(* IEC 61131-3 sources: ElnaAutomator/ExampleProject/build_USO_ecl, 1 file *)

(* ---- plc.st ---- *)
TYPE
  struct_singleOutput : STRUCT
    wait_time : TIME;
    inCommand : WORD;
    inOpcCommandsDisabled : BOOL;
    Q : BOOL;
    status : DWORD;
    OpcCommandsDisabled : BOOL;
    inCommand_Alg : WORD;
    inCommand_ARM : WORD;
  END_STRUCT;
  Im_singleOutputs : STRUCT
    So0 : struct_singleOutput;
    So1 : struct_singleOutput;
    So2 : struct_singleOutput;
    So3 : struct_singleOutput;
    So4 : struct_singleOutput;
    So5 : struct_singleOutput;
    So6 : struct_singleOutput;
    So7 : struct_singleOutput;
  END_STRUCT;
  struct_SectionSwitch : STRUCT
    inCommand : WORD;
    status : DWORD;
    onStatus : BYTE;
    inOpcCommandsDisabled : BOOL;
    sdvig : BOOL;
    Ns : BOOL;
    CommandFault : BOOL;
    Accident : BOOL;
    Local : BOOL;
    Distance : BOOL;
    OpcCommandsDisabled : BOOL;
    lastCmdIsOn : BOOL;
    offKNA : BOOL;
    basketStatus : BYTE;
    ISVALIDREF_statOn : BOOL;
    ISVALIDREF_statOff : BOOL;
    ISVALIDREF_cmdOn : BOOL;
    ISVALIDREF_cmdOff : BOOL;
    ISVALIDREF_inBreakCmdOn : BOOL;
    ISVALIDREF_inBreakCmdOff : BOOL;
    BreakCmdOn : BOOL;
    BreakCmdOff : BOOL;
    ISVALIDREF_basketRolledIn : BOOL;
    ISVALIDREF_basketRolledOut : BOOL;
    ISVALIDREF_basketTest : BOOL;
    inCommand_Alg : WORD;
    inCommand_ARM : WORD;
    cmdOn : BOOL;
    cmdOff : BOOL;
    reliability : BOOL;
  END_STRUCT;
  TYPE_ReliableBit : STRUCT
    value : BOOL;
    reliability : BOOL;
    _inversed : BOOL;
  END_STRUCT;
  struct_DI : STRUCT
    imit : BOOL;
    value : WORD;
    reliability : WORD;
    bits : ARRAY [0..15] OF TYPE_ReliableBit;
    blConnect : BOOL;
  END_STRUCT;
  DiConfig : STRUCT
    Di : struct_DI;
    Di1 : struct_DI;
    Di2 : struct_DI;
    Di3 : struct_DI;
    Di4 : struct_DI;
  END_STRUCT;
  TYPE_ProtectionTags : STRUCT
    NOTHING : BYTE := 0;
    AOB : BYTE := 1;
    AOS : BYTE := 2;
    AOPOJ : BYTE := 3;
  END_STRUCT;
  struct_singleSignal : STRUCT
    reliability : BOOL;
    inverse : BOOL;
    DelayOn : TIME;
    DelayOff : TIME;
    Q : BOOL;
    status : DWORD;
    Disabled_Sig : BOOL;
  END_STRUCT;
  struct_AiProtection : STRUCT
    controlLimit : BYTE;
    delay : TIME;
    inTag : BYTE;
    inRunOnStart : BOOL;
    inCanRun : BOOL;
    inOpcCommandsDisabled : BOOL;
    inCommand : WORD;
    inCommand_Alg : WORD;
    inCommand_ARM : WORD;
    Tag : BYTE;
    status : DWORD;
    CanRun : BOOL;
    OpcCommandsDisabled : BOOL;
    isRunning : BOOL;
    HasError : BOOL;
    isEnded : BOOL;
    Remont : BOOL;
    Check : BOOL;
    Signaling : BOOL;
    SignalingTP : BOOL;
    RunOnStart : BOOL;
  END_STRUCT;
  TDoubleData : STRUCT
    wFlags : UINT := 0;
    dblValue : LREAL := 0.0;
  END_STRUCT;
  struct_DO : STRUCT
    imit : BOOL;
    blConnect : BOOL;
    value : WORD;
    bits : ARRAY [0..15] OF BOOL;
  END_STRUCT;
  DoConfig : STRUCT
    Do1 : struct_DO;
    Do2 : struct_DO;
    Do3 : struct_DO;
    Do4 : struct_DO;
    Do5 : struct_DO;
  END_STRUCT;
  struct_ReserveIM2 : STRUCT
    var1 : BOOL;
    var2 : BOOL;
  END_STRUCT;
  struct_Kran : STRUCT
    inCommand : WORD;
    status : DWORD;
    onStatus : BYTE;
    inOpcCommandsDisabled : BOOL;
    sdvig : BOOL;
    Ns : BOOL;
    Dp : BOOL;
    CommandFault : BOOL;
    Accident : BOOL;
    Auto : BOOL;
    Manual : BOOL;
    Local : BOOL;
    Distance : BOOL;
    ErrorPowerOff : BOOL;
    ErrorBlock : BOOL;
    So : BOOL;
    Sz : BOOL;
    OpcCommandsDisabled : BOOL;
    lastCmdIsOn : BOOL;
    ISVALIDREF_statOn : BOOL;
    ISVALIDREF_statOff : BOOL;
    ISVALIDREF_cmdOn : BOOL;
    ISVALIDREF_cmdOff : BOOL;
    ISVALIDREF_inSo : BOOL;
    ISVALIDREF_inSz : BOOL;
    ISVALIDREF_inDp : BOOL;
    continueHoldCommand : TIME;
    inCommand_Alg : WORD;
    inCommand_ARM : WORD;
    cmdOn : BOOL;
    cmdOff : BOOL;
    reliability : BOOL;
  END_STRUCT;
  struct_OilPump : STRUCT
    inCommand : WORD;
    inCommand_Alg : WORD;
    inCommand_ARM : WORD;
    status : DWORD;
    onStatus : BYTE;
    inOpcCommandsDisabled : BOOL;
    sdvig : BOOL;
    Ns : BOOL;
    CommandFault : BOOL;
    Accident : BOOL;
    Local : BOOL;
    Distance : BOOL;
    BreakCmdOn : BOOL;
    BreakCmdOff : BOOL;
    OpcCommandsDisabled : BOOL;
    lastCmdIsOn : BOOL;
    ISVALIDREF_statOn : BOOL;
    ISVALIDREF_statOff : BOOL;
    ISVALIDREF_cmdOn : BOOL;
    ISVALIDREF_cmdOff : BOOL;
    ISVALIDREF_inBreakCmdOn : BOOL;
    ISVALIDREF_inBreakCmdOff : BOOL;
    inBlocked : BOOL;
    Blocked : BOOL;
    Osnovnoy : BOOL;
    Rezervny : BOOL;
    cmdOn : BOOL;
    cmdOff : BOOL;
    reliability : BOOL;
  END_STRUCT;
  struct_Switch : STRUCT
    inCommand : WORD;
    status : DWORD;
    onStatus : BYTE;
    inOpcCommandsDisabled : BOOL;
    sdvig : BOOL;
    Ns : BOOL;
    CommandFault : BOOL;
    Accident : BOOL;
    Auto : BOOL;
    Manual : BOOL;
    Local : BOOL;
    Distance : BOOL;
    ErrorPowerOff : BOOL;
    ErrorBlock : BOOL;
    BreakCmdOn : BOOL;
    BreakCmdOff : BOOL;
    OpcCommandsDisabled : BOOL;
    lastCmdIsOn : BOOL;
    ISVALIDREF_statOn : BOOL;
    ISVALIDREF_statOff : BOOL;
    ISVALIDREF_cmdOn : BOOL;
    ISVALIDREF_cmdOff : BOOL;
    ISVALIDREF_inBreakCmdOn : BOOL;
    ISVALIDREF_inBreakCmdOff : BOOL;
    inCommand_Alg : WORD;
    inCommand_ARM : WORD;
    cmdOn : BOOL;
    cmdOff : BOOL;
    reliability : BOOL;
  END_STRUCT;
  Im_singleSignals : STRUCT
    SI0 : struct_singleSignal;
    SI1 : struct_singleSignal;
    SI2 : struct_singleSignal;
    SI3 : struct_singleSignal;
    SI4 : struct_singleSignal;
    SI5 : struct_singleSignal;
    SI6 : struct_singleSignal;
  END_STRUCT;
  ImConfig : STRUCT
    Kran1 : struct_Kran;
    Kran4 : struct_Kran;
    Kran2 : struct_Kran;
    Kran3 : struct_Kran;
    Nu : struct_OilPump;
    Nu2 : struct_OilPump;
    Avom1 : struct_Switch;
    Avom2 : struct_Switch;
    Avom3 : struct_Switch;
    Avom4 : struct_Switch;
    Mv : struct_SectionSwitch;
    SectionSwitch1 : struct_SectionSwitch;
    SingleSignals : Im_singleSignals;
    SingleOutputs : Im_singleOutputs;
  END_STRUCT;
  struct_DiProtection : STRUCT
    delay : TIME;
    inTag : BYTE;
    inRunOnStart : BOOL;
    inCanRun : BOOL;
    inOpcCommandsDisabled : BOOL;
    inCommand : WORD;
    inCommand_Alg : WORD;
    inCommand_ARM : WORD;
    Tag : BYTE;
    status : DWORD;
    CanRun : BOOL;
    OpcCommandsDisabled : BOOL;
    isRunning : BOOL;
    HasError : BOOL;
    isEnded : BOOL;
    Remont : BOOL;
    Check : BOOL;
    Signaling : BOOL;
    SignalingTP : BOOL;
    RunOnStart : BOOL;
  END_STRUCT;
  ProtectionsConfig : STRUCT
    Ap1 : struct_AiProtection;
    AiP1 : struct_AiProtection;
    AiP2 : struct_AiProtection;
    AiP3 : struct_AiProtection;
    DiP1 : struct_DiProtection;
    DiP2 : struct_DiProtection;
    DiP3 : struct_DiProtection;
    DiP4 : struct_DiProtection;
    DiP5 : struct_DiProtection;
  END_STRUCT;
  TYPE_StatusAi : STRUCT
    NOTDEFINED : BYTE := 0;
    LL : BYTE := 1;
    HL : BYTE := 2;
    NOTRELIABLE : BYTE := 3;
    normal : BYTE := 4;
    LW : BYTE := 5;
    HW : BYTE := 6;
    LA : BYTE := 7;
    HA : BYTE := 8;
  END_STRUCT;
  TItemAIN : STRUCT
    wFlags : UINT := 0;
    wReserved : UINT := 0;
    dblValue : LREAL := 0.0;
    nanosec : ULINT := 0;
    reserve : ULINT := 0;
  END_STRUCT;
  TItemDIN : STRUCT
    wFlags : UINT := 0;
    wValue : UINT := 0;
    nanosec : ULINT := 0;
    reserve : ULINT := 0;
  END_STRUCT;
  struct_AI : STRUCT
    value : LREAL;
    status : DWORD;
    interval : BYTE;
    inCommand : WORD;
    blConnect : BOOL;
    dLL : LREAL;
    dHL : LREAL;
    dLA : LREAL;
    dHA : LREAL;
    dLW : LREAL;
    dHW : LREAL;
    LL : LREAL;
    HL : LREAL;
    LA : LREAL;
    HA : LREAL;
    LW : LREAL;
    HW : LREAL;
    ISVALIDREF_LA : BOOL;
    ISVALIDREF_HA : BOOL;
    ISVALIDREF_LW : BOOL;
    ISVALIDREF_HW : BOOL;
    inpLL : LREAL;
    inpHL : LREAL;
    CurrentShotCircuit : LREAL;
    CurrentBreakCircuit : LREAL;
    maxChangeSpeed : LREAL;
    maxChangeSpeedDown : LREAL;
    ChangeSpeed : LREAL;
    histeresis : LREAL;
    aperturFilter : LREAL;
    exponentialFilter : LREAL;
    rassoglasovanie : LREAL;
    OpcCommandsDisabled : BOOL;
    Disabled_LA : BOOL;
    Disabled_HA : BOOL;
    Disabled_LW : BOOL;
    Disabled_HW : BOOL;
    delayLA : TIME;
    delayLW : TIME;
    delayHW : TIME;
    delayHA : TIME;
    minValue_ISVALIDREF : BOOL;
    maxValue_ISVALIDREF : BOOL;
    minValue : LREAL;
    maxValue : LREAL;
    inOpcCommandsDisabled : BOOL;
    imit : BOOL;
    remont : BOOL;
    NS : BOOL;
    NS_Min : BOOL;
    NS_Max : BOOL;
    inCommand_Alg : WORD;
    inCommand_ARM : WORD;
  END_STRUCT;
  AiConfig : STRUCT
    A1 : struct_AI;
    A2 : struct_AI;
  END_STRUCT;
  TWordData : STRUCT
    wFlags : UINT := 0;
    wValue : UINT := 0;
  END_STRUCT;
  TYPE_statusDualInput : STRUCT
    STATUS_NOTDEFINED : BYTE := 0;
    STATUS_ON : BYTE := 1;
    STATUS_OFF : BYTE := 2;
    STATUS_TRANSITIONAL : BYTE := 3;
    STATUS_ERROR : BYTE := 4;
  END_STRUCT;
  TYPE_AnalogLimitFlags : STRUCT
    NONE : BYTE := 0;
    LL : BYTE := 16#1;
    LW : BYTE := 16#2;
    HW : BYTE := 16#4;
    LA : BYTE := 16#8;
    HA : BYTE := 16#10;
    HL : BYTE := 16#20;
  END_STRUCT;
  TYPE_basketStats : STRUCT
    BASKET_NOTDEFINED : BYTE := 0;
    BASKET_ROLLEDIN : BYTE := 1;
    BASKET_ROLLEDOUT : BYTE := 2;
    BASKET_TRANSITIONAL : BYTE := 3;
    BASKET_ERROR : BYTE := 4;
    BASKET_TEST : BYTE := 5;
  END_STRUCT;
  TYPE_CommandAnalog : STRUCT
    cmd_SetUstavki : WORD := 1;
    cmd_SetRemont : WORD := 2;
    cmd_ResetRemont : WORD := 3;
    cmd_kvitNotReliable : WORD := 4;
  END_STRUCT;
  TYPE_commandDualInput : STRUCT
    CMD_ON : BYTE := 1;
    CMD_OFF : BYTE := 2;
    CMD_RESET : BYTE := 3;
  END_STRUCT;
  struct_ReserveIM : STRUCT
    var1 : BOOL;
    var2 : BOOL;
  END_STRUCT;
  struct_DiscretParametr : STRUCT
    newValue : UINT;
    currentValue : UINT;
    inOpcCommandsDisabled : BOOL;
    inCommand : WORD;
    inCommand_Alg : WORD;
    inCommand_ARM : WORD;
    status : DWORD;
    OpcCommandsDisabled : BOOL;
    Value : UINT;
  END_STRUCT;
END_TYPE

FUNCTION UnBlockAllIm : BOOL
  VAR_IN_OUT
    IM : ImConfig;
  END_VAR

  IF IM.Kran1.inOpcCommandsDisabled THEN IM.Kran1.inOpcCommandsDisabled := FALSE; END_IF;
  IF IM.Kran4.inOpcCommandsDisabled THEN IM.Kran4.inOpcCommandsDisabled := FALSE; END_IF;
  IF IM.Kran2.inOpcCommandsDisabled THEN IM.Kran2.inOpcCommandsDisabled := FALSE; END_IF;
  IF IM.Kran3.inOpcCommandsDisabled THEN IM.Kran3.inOpcCommandsDisabled := FALSE; END_IF;
  IF IM.Nu.inOpcCommandsDisabled THEN IM.Nu.inOpcCommandsDisabled := FALSE; END_IF;
  IF IM.Nu2.inOpcCommandsDisabled THEN IM.Nu2.inOpcCommandsDisabled := FALSE; END_IF;
  IF IM.Avom1.inOpcCommandsDisabled THEN IM.Avom1.inOpcCommandsDisabled := FALSE; END_IF;
  IF IM.Avom2.inOpcCommandsDisabled THEN IM.Avom2.inOpcCommandsDisabled := FALSE; END_IF;
  IF IM.Avom3.inOpcCommandsDisabled THEN IM.Avom3.inOpcCommandsDisabled := FALSE; END_IF;
  IF IM.Avom4.inOpcCommandsDisabled THEN IM.Avom4.inOpcCommandsDisabled := FALSE; END_IF;
  IF IM.Mv.inOpcCommandsDisabled THEN IM.Mv.inOpcCommandsDisabled := FALSE; END_IF;
  IF IM.SectionSwitch1.inOpcCommandsDisabled THEN IM.SectionSwitch1.inOpcCommandsDisabled := FALSE; END_IF;
END_FUNCTION

FUNCTION TwoUint_To_UDINT : UDINT
  VAR_INPUT
    val1 : UINT;
    val2 : UINT;
  END_VAR

  TwoUint_To_UDINT:= DWORD_TO_UDINT(UINT_TO_DWORD(val1) OR shl(UINT_TO_DWORD(val2), 16));
END_FUNCTION

FUNCTION BlockAllProtections : BOOL
  VAR_IN_OUT
    Protections : ProtectionsConfig;
  END_VAR

  Protections.Ap1.inOpcCommandsDisabled := TRUE;
  Protections.AiP1.inOpcCommandsDisabled := TRUE;
  Protections.AiP2.inOpcCommandsDisabled := TRUE;
  Protections.AiP3.inOpcCommandsDisabled := TRUE;
  Protections.DiP1.inOpcCommandsDisabled := TRUE;
  Protections.DiP2.inOpcCommandsDisabled := TRUE;
  Protections.DiP3.inOpcCommandsDisabled := TRUE;
  Protections.DiP4.inOpcCommandsDisabled := TRUE;
  Protections.DiP5.inOpcCommandsDisabled := TRUE;
END_FUNCTION

FUNCTION BlockAllIm : BOOL
  VAR_IN_OUT
    IM : ImConfig;
  END_VAR

  IF NOT IM.Kran1.inOpcCommandsDisabled THEN IM.Kran1.inOpcCommandsDisabled := TRUE; END_IF;
  IF NOT IM.Kran4.inOpcCommandsDisabled THEN IM.Kran4.inOpcCommandsDisabled := TRUE; END_IF;
  IF NOT IM.Kran2.inOpcCommandsDisabled THEN IM.Kran2.inOpcCommandsDisabled := TRUE; END_IF;
  IF NOT IM.Kran3.inOpcCommandsDisabled THEN IM.Kran3.inOpcCommandsDisabled := TRUE; END_IF;
  IF NOT IM.Nu.inOpcCommandsDisabled THEN IM.Nu.inOpcCommandsDisabled := TRUE; END_IF;
  IF NOT IM.Nu2.inOpcCommandsDisabled THEN IM.Nu2.inOpcCommandsDisabled := TRUE; END_IF;
  IF NOT IM.Avom1.inOpcCommandsDisabled THEN IM.Avom1.inOpcCommandsDisabled := TRUE; END_IF;
  IF NOT IM.Avom2.inOpcCommandsDisabled THEN IM.Avom2.inOpcCommandsDisabled := TRUE; END_IF;
  IF NOT IM.Avom3.inOpcCommandsDisabled THEN IM.Avom3.inOpcCommandsDisabled := TRUE; END_IF;
  IF NOT IM.Avom4.inOpcCommandsDisabled THEN IM.Avom4.inOpcCommandsDisabled := TRUE; END_IF;
  IF NOT IM.Mv.inOpcCommandsDisabled THEN IM.Mv.inOpcCommandsDisabled := TRUE; END_IF;
  IF NOT IM.SectionSwitch1.inOpcCommandsDisabled THEN IM.SectionSwitch1.inOpcCommandsDisabled := TRUE; END_IF;
END_FUNCTION

FUNCTION resetAiProtection : BOOL
  VAR_IN_OUT
    protection : struct_AiProtection;
  END_VAR
  VAR CONSTANT
    cmdReset : WORD    := 2;
  END_VAR

  IF protection.isRunning THEN
                      protection.inOpcCommandsDisabled:=TRUE;
  		protection.inCommand_Alg:=cmdReset;
  END_IF;
END_FUNCTION

FUNCTION resetDiProtection : BOOL
  VAR_IN_OUT
    protection : struct_DiProtection;
  END_VAR
  VAR CONSTANT
    cmdReset : WORD    := 2;
  END_VAR

  IF protection.isRunning THEN
                      protection.inOpcCommandsDisabled:=TRUE;
  		protection.inCommand_Alg:=cmdReset;
  END_IF;
END_FUNCTION

FUNCTION ResetAllProtections : BOOL
  VAR_IN_OUT
    Protections : ProtectionsConfig;
  END_VAR

  ResetAiProtection(Protections.Ap1);
  ResetAiProtection(Protections.AiP1);
  ResetAiProtection(Protections.AiP2);
  ResetAiProtection(Protections.AiP3);
  ResetDiProtection(Protections.DiP1);
  ResetDiProtection(Protections.DiP2);
  ResetDiProtection(Protections.DiP3);
  ResetDiProtection(Protections.DiP4);
  ResetDiProtection(Protections.DiP5);
END_FUNCTION

FUNCTION ResetAllSignaling : BOOL
  VAR_IN_OUT
    Protections : ProtectionsConfig;
  END_VAR

  IF Protections.Ap1.Signaling THEN
  	ResetAiProtection(Protections.Ap1); END_IF;
  IF Protections.AiP1.Signaling THEN
  	ResetAiProtection(Protections.AiP1); END_IF;
  IF Protections.AiP2.Signaling THEN
  	ResetAiProtection(Protections.AiP2); END_IF;
  IF Protections.AiP3.Signaling THEN
  	ResetAiProtection(Protections.AiP3); END_IF;
  IF Protections.DiP1.Signaling THEN
  	ResetDiProtection(Protections.DiP1); END_IF;
  IF Protections.DiP2.Signaling THEN
  	ResetDiProtection(Protections.DiP2); END_IF;
  IF Protections.DiP3.Signaling THEN
  	ResetDiProtection(Protections.DiP3); END_IF;
  IF Protections.DiP4.Signaling THEN
  	ResetDiProtection(Protections.DiP4); END_IF;
  IF Protections.DiP5.Signaling THEN
  	ResetDiProtection(Protections.DiP5); END_IF;
END_FUNCTION

FUNCTION AnyAnalogsPs : BOOL
  VAR_INPUT
    Ai : AiConfig;
  END_VAR
  VAR
    statusAi : TYPE_StatusAi;
  END_VAR

  AnyAnalogsPs :=
  Ai.A1.interval = statusAi.HW OR
  Ai.A2.interval = statusAi.HW OR
  Ai.A1.interval = statusAi.LW OR
  Ai.A2.interval = statusAi.LW;
END_FUNCTION

FUNCTION AnyAnalogsNs : BOOL
  VAR_INPUT
    Ai : AiConfig;
  END_VAR
  VAR
    statusAi : TYPE_StatusAi;
  END_VAR

  AnyAnalogsNs :=
  ((Ai.A1.interval < statusAi.Normal) AND NOT Ai.A1.Remont) OR
  ((Ai.A2.interval < statusAi.Normal) AND NOT Ai.A2.Remont);
END_FUNCTION

FUNCTION NsCepeiControl : BOOL
  VAR_INPUT
    IM : ImConfig;
  END_VAR

  NsCepeiControl := NOT (
  	IM.Kran1.reliability OR
  	IM.Kran4.reliability OR
  	IM.Kran2.reliability OR
  	IM.Kran3.reliability OR
  	IM.Nu.reliability OR
  	IM.Nu2.reliability OR
  	IM.Avom1.reliability OR
  	IM.Avom2.reliability OR
  	IM.Avom3.reliability OR
  	IM.Avom4.reliability OR
  	IM.Mv.reliability OR
  	IM.SectionSwitch1.reliability);
END_FUNCTION

FUNCTION EnableAiLimits : BOOL
  VAR_IN_OUT
    Ai : AiConfig;
  END_VAR

  Ai.A1.Disabled_LA := FALSE;
  Ai.A2.Disabled_LA := FALSE;
  Ai.A1.Disabled_LW := FALSE;
  Ai.A2.Disabled_LW := FALSE;
END_FUNCTION

FUNCTION AnyDiscretPs : BOOL
  VAR_INPUT
    Im : ImConfig;
  END_VAR

  AnyDiscretPs :=
  Im.SingleSignals.SI0.Q;
END_FUNCTION

FUNCTION AnyDiscretNs : BOOL
  VAR_INPUT
    Di : DiConfig;
  END_VAR

  AnyDiscretNs :=
  ((Di.Di.reliability <> 255) OR
  (Di.Di1.reliability <> 255) OR
  (Di.Di2.reliability <> 255) OR
  (Di.Di3.reliability <> 255) OR
  (Di.Di4.reliability <> 255));
END_FUNCTION

FUNCTION UnBlockAllProtections : BOOL
  VAR_IN_OUT
    Protections : ProtectionsConfig;
  END_VAR

  protections.Ap1.inOpcCommandsDisabled := FALSE;
  protections.AiP1.inOpcCommandsDisabled := FALSE;
  protections.AiP2.inOpcCommandsDisabled := FALSE;
  protections.AiP3.inOpcCommandsDisabled := FALSE;
  protections.DiP1.inOpcCommandsDisabled := FALSE;
  protections.DiP2.inOpcCommandsDisabled := FALSE;
  protections.DiP3.inOpcCommandsDisabled := FALSE;
  protections.DiP4.inOpcCommandsDisabled := FALSE;
  protections.DiP5.inOpcCommandsDisabled := FALSE;
END_FUNCTION

FUNCTION AnyProtectionSignaling : BOOL
  VAR_INPUT
    Protections : ProtectionsConfig;
  END_VAR

  AnyProtectionSignaling :=
  Protections.Ap1.Signaling OR
  Protections.AiP1.Signaling OR
  Protections.AiP2.Signaling OR
  Protections.AiP3.Signaling OR
  Protections.DiP1.Signaling OR
  Protections.DiP2.Signaling OR
  Protections.DiP3.Signaling OR
  Protections.DiP4.Signaling OR
  Protections.DiP5.Signaling;
END_FUNCTION

FUNCTION AnyProtectionInRemont : BOOL
  VAR_INPUT
    Protections : ProtectionsConfig;
  END_VAR

  AnyProtectionInRemont :=
  Protections.Ap1.Remont OR
  Protections.AiP1.Remont OR
  Protections.AiP2.Remont OR
  Protections.AiP3.Remont OR
  Protections.DiP1.Remont OR
  Protections.DiP2.Remont OR
  Protections.DiP3.Remont OR
  Protections.DiP4.Remont OR
  Protections.DiP5.Remont;
END_FUNCTION

FUNCTION runDiProtection : BOOL
  VAR_IN_OUT
    protection : struct_DiProtection;
  END_VAR
  VAR CONSTANT
    cmdRun : WORD    := 1;
  END_VAR

  IF NOT protection.isRunning THEN
                      protection.inOpcCommandsDisabled:=TRUE;
  		protection.inCommand_Alg:=cmdRun;
  END_IF;
END_FUNCTION

FUNCTION runAiProtection : BOOL
  VAR_IN_OUT
    protection : struct_AiProtection;
  END_VAR
  VAR CONSTANT
    cmdRun : WORD    := 1;
  END_VAR

  IF NOT protection.isRunning THEN
                      protection.inOpcCommandsDisabled:=TRUE;
  		protection.inCommand_Alg:=cmdRun;
  END_IF;
END_FUNCTION

FUNCTION AutoRunProtections : BOOL
  VAR_IN_OUT
    Protections : ProtectionsConfig;
  END_VAR

  RunAiProtection(Protections.Ap1);
  RunAiProtection(Protections.AiP2);
  RunDiProtection(Protections.DiP1);
  RunDiProtection(Protections.DiP2);
  RunDiProtection(Protections.DiP3);
END_FUNCTION

FUNCTION DIwValue_Diag : UDINT
  VAR_INPUT
    val1 : UINT;
    val2 : UINT;
  END_VAR
  VAR
    val1_tmp : DWORD;
    val2_tmp : DWORD;
  END_VAR

  (* Переставлем биты value и reability местами для корректного отображения в MasterScada *)

  val1_tmp:=(SHL(UINT_TO_DWORD(val1),1) AND 16#AAAA) OR (SHR(UINT_TO_DWORD(val1),1) AND 16#5555);

  val2_tmp:=(SHL(UINT_TO_DWORD(val2),1) AND 16#AAAA) OR (SHR(UINT_TO_DWORD(val2),1) AND 16#5555);

  (* Вместо reability = 1 посдставляем инверсию сигнала в виде , если нет reability тогда обрыв = 1 для MasterScada *)

  DIwValue_Diag:= DWORD_TO_UDINT((val1_tmp OR shl(val2_tmp, 16)) XOR 16#55555555);
END_FUNCTION

FUNCTION DisableAiLimits : BOOL
  VAR_IN_OUT
    Ai : AiConfig;
  END_VAR

  Ai.A1.Disabled_LA := TRUE;
  Ai.A2.Disabled_LA := TRUE;
  Ai.A1.Disabled_LW := TRUE;
  Ai.A2.Disabled_LW := TRUE;
END_FUNCTION

FUNCTION RemontAllProtections : BOOL
  VAR_IN_OUT
    Protections : ProtectionsConfig;
  END_VAR
  VAR CONSTANT
    cmdRemont : WORD  := 4;
  END_VAR

  Protections.Ap1.inCommand_Alg := cmdRemont;
  Protections.AiP1.inCommand_Alg := cmdRemont;
  Protections.AiP2.inCommand_Alg := cmdRemont;
  Protections.AiP3.inCommand_Alg := cmdRemont;
  Protections.DiP1.inCommand_Alg := cmdRemont;
  Protections.DiP2.inCommand_Alg := cmdRemont;
  Protections.DiP3.inCommand_Alg := cmdRemont;
  Protections.DiP4.inCommand_Alg := cmdRemont;
  Protections.DiP5.inCommand_Alg := cmdRemont;
END_FUNCTION

FUNCTION NsCepeiUpravlenya : BOOL
  VAR_INPUT
    IM : ImConfig;
  END_VAR

  NsCepeiUpravlenya := (
  	IM.Kran4.Sz OR
  	IM.Kran2.Sz OR
  	IM.Kran3.So OR
  	IM.Nu.breakCmdOn OR
  	IM.Nu2.breakCmdOn OR
  	IM.Avom1.breakCmdOn OR
  	IM.Avom2.breakCmdOn OR
  	IM.Avom3.breakCmdOn OR
  	IM.Avom4.breakCmdOn OR
  	IM.Mv.breakCmdOn);
END_FUNCTION

FUNCTION_BLOCK fb_DOSourceMlp
  VAR_IN_OUT
    arDout : TWordData;
  END_VAR
  VAR_INPUT
    err_mod : TItemDIN;
  END_VAR
  VAR_IN_OUT
    strDO : struct_DO;
  END_VAR
  VAR
    bitNumber : INT;
  END_VAR

  strDO.blConnect := ((UINT_TO_WORD(err_mod.wValue) = 20) and (UINT_TO_WORD(err_mod.wFlags) = 192));

  strDO.value:=0;

  FOR bitNumber:=0 TO 15 BY 1 DO
  	strDO.value:=strDO.value OR (SHL(BOOL_TO_WORD(strDO.bits[bitNumber]),bitNumber));
  END_FOR;

  IF NOT strDO.imit THEN
  	 arDout.wValue:= WORD_TO_UINT(strDO.value);
  END_IF;
END_FUNCTION_BLOCK

FUNCTION_BLOCK fb_DI_Init
  VAR_INPUT
    data_Ini : BOOL;
    imit : BOOL    := FALSE;
  END_VAR
  VAR_IN_OUT
    strDI : struct_DI;
  END_VAR
  VAR_OUTPUT
    Init : BOOL    := FALSE;
  END_VAR

  (*****            Функциональный блок переинициализации структуры-дескриптора канала дискретного ввода        *****)

   Init := FALSE;

      IF data_Ini THEN                            (* Параметрам требуется переинициализация. *)
          strDI.imit       := imit;
          data_Ini:=FALSE;
          Init := TRUE;
      END_IF;
    IF Init THEN
  imit:=FALSE;
      END_IF;
END_FUNCTION_BLOCK

FUNCTION_BLOCK fb_sunpackerCommand
  VAR_INPUT
    command : WORD;
  END_VAR
  VAR_OUTPUT
    source : BYTE;
    parametr : BYTE;
    cmd : BYTE;
  END_VAR

  cmd := WORD_TO_BYTE(command and 16#7);
  parametr := WORD_TO_BYTE(SHR((command and 16#1FF8), 3));
  source := WORD_TO_BYTE(SHR(command, 13));
END_FUNCTION_BLOCK

FUNCTION_BLOCK fb_Switch
  VAR_INPUT
    statOn : BOOL;
    statOff : BOOL;
    statOn_reliability : BOOL;
    statOff_reliability : BOOL;
  END_VAR
  VAR_IN_OUT
    StrSw : struct_Switch;
  END_VAR
  VAR_INPUT
    inNs : TYPE_ReliableBit;
    inAccident : TYPE_ReliableBit;
    inAuto : TYPE_ReliableBit;
    inManual : TYPE_ReliableBit;
    inLocal : TYPE_ReliableBit;
    inDistance : TYPE_ReliableBit;
    inErrorPowerOff : TYPE_ReliableBit;
    inErrorBlock : TYPE_ReliableBit;
    inBreakCmdOn : TYPE_ReliableBit;
    inBreakCmdOff : TYPE_ReliableBit;
  END_VAR
  VAR
    onInit : BOOL    := FALSE;
    _statOn : BOOL;
    _statOff : BOOL;
    lastOnStatus : BYTE;
    cmd : BYTE;
    source : BYTE;
    lastCmd : BYTE;
    source_for_Status : BYTE;
    cmd_for_Status : BYTE;
    command_error_for_Status : BYTE;
    _sunpackerCommand : fb_sunpackerCommand;
    _statusDualInput : TYPE_statusDualInput;
    _commandDualInput : TYPE_commandDualInput;
    _commandErrorTimer : BOOL;
    resetErrorTimer : BOOL;
    getSdvig : BOOL;
    _changWithoutCommand : BOOL;
    errorCMDTimer : TON;
    sdvigReset : TON;
    _errorReset : TON;
    outputsSets : TOF;
  END_VAR
  VAR_IN_OUT
    cmdOn : BOOL;
    cmdOff : BOOL;
  END_VAR

  IF NOT onInit THEN
  IF StrSw.ISVALIDREF_cmdOn XOR StrSw.ISVALIDREF_cmdOff THEN
  	IF 	StrSw.ISVALIDREF_cmdOn THEN
  		lastCmd:= 2; (*baseCmdOff*)
  	ELSE
  		lastCmd:= 1; (*baseCmdOn*)
  	END_IF;
  END_IF;
  onInit:=TRUE;
  END_IF;

  (* ---- Если управление с ВУ заблокировано, то в ИМ передаем команду из алгоритма ---- *)
  IF StrSw.inOpcCommandsDisabled THEN
  	StrSw.inCommand := StrSw.inCommand_Alg;
  ELSE (* иначе передаем команду с АРМа*)
  	StrSw.inCommand := StrSw.inCommand_ARM;
  END_IF;

  (* ---- Формирование состояния механизма ---- *)

  IF (StrSw.ISVALIDREF_statOn) OR (StrSw.ISVALIDREF_statOff) THEN
  	IF (StrSw.ISVALIDREF_statOn) AND (StrSw.ISVALIDREF_statOff) THEN
  	StrSw.reliability:= statOn_reliability AND statOff_reliability;
  		_statOn  := statOn;
  		_statOff := statOff;
  	ELSIF (StrSw.ISVALIDREF_statOn) THEN
                       StrSw.reliability:= statOn_reliability;
  		_statOn  := statOn;
  		_statOff := NOT statOn;
  	ELSIF (StrSw.ISVALIDREF_statOff) THEN
  		 StrSw.reliability:= statOff_reliability;
  		_statOn  := NOT statOff;
  		_statOff :=statOff;
  	END_IF;

  	IF StrSw.reliability THEN
  		IF _statOn AND NOT _statOff 		THEN 	StrSw.onStatus := _statusDualInput.STATUS_ON;
  		ELSIF _statOff AND NOT _statOn 	THEN 	StrSw.onStatus := _statusDualInput.Status_OFF;
  		ELSIF NOT _statOn AND NOT _statOff 	THEN 	StrSw.onStatus := _statusDualInput.STATUS_TRANSITIONAL;
  		ELSE					StrSw.onStatus := _statusDualInput.STATUS_ERROR;
                      END_IF;

  	ELSE
  		StrSw.onStatus := _statusDualInput.STATUS_NOTDEFINED;

  	END_IF;
  ELSE
  	CASE BYTE_TO_INT(lastCmd) OF
  		(*baseCmdOn*) 1: StrSw.onStatus  := _statusDualInput.STATUS_ON;
  		(*baseCmdOff*) 2: StrSw.onStatus  := _statusDualInput.STATUS_OFF;

  	ELSE
  		 StrSw.onStatus := _statusDualInput.STATUS_NOTDEFINED;

  	END_CASE;
  END_IF;

  StrSw.Accident := inAccident.value AND inAccident.reliability;
  StrSw.Ns := inNs.value AND inNs.reliability;
  StrSw.Auto := inAuto.value AND inAuto.reliability;
  StrSw.Manual := inManual.value AND inManual.reliability;
  StrSw.Local := inLocal.value AND inLocal.reliability;
  StrSw.Distance := inDistance.value AND inDistance.reliability;
  StrSw.ErrorPowerOff := inErrorPowerOff.value AND inErrorPowerOff.reliability;
  StrSw.ErrorBlock := inErrorBlock.value AND inErrorBlock.reliability;
  StrSw.OpcCommandsDisabled := StrSw.inOpcCommandsDisabled;

  (* ---- Формирование признака сдвига ---- *)
  getSdvig := FALSE;
  IF (StrSw.ISVALIDREF_cmdOn OR StrSw.ISVALIDREF_cmdOff) AND NOT StrSw.Local THEN
  	IF NOT (StrSw.CmdOn OR StrSw.CmdOff) THEN
                       IF (lastOnStatus <> StrSw.onStatus AND
  		(StrSw.onStatus <> _statusDualInput.STATUS_NOTDEFINED AND
                       StrSw.onStatus <> _statusDualInput.STATUS_ERROR)     AND
  		(lastOnStatus <> _statusDualInput.STATUS_NOTDEFINED   AND
                       lastOnStatus <> _statusDualInput.STATUS_ERROR))
                      THEN
  			getSdvig   := TRUE;
  		END_IF;
  	END_IF;
  END_IF;

  IF getSdvig THEN StrSw.sdvig:= TRUE; END_IF;

  sdvigReset(IN:=StrSw.sdvig, PT:=T#15S);

  IF sdvigReset.Q THEN StrSw.sdvig:=FALSE; END_IF;

  lastOnStatus := StrSw.onStatus;

  (* ---- Распаковка команды ---- *)
  _sunpackerCommand(command := StrSw.inCommand);
  	cmd := _sunpackerCommand.cmd;
  	source := _sunpackerCommand.source;

  (* ---- Обработка команды ---- *)
  IF cmd <> 0 AND lastCmd <> cmd and (((NOT StrSw.opcCommandsDisabled) AND source > 0) OR source = 0) then
  	CASE BYTE_TO_INT(cmd) OF
  	(*cmd_open*) 1 :
  			IF  StrSw.ISVALIDREF_cmdOn THEN StrSw.CmdOn := TRUE;
  				IF StrSw.ISVALIDREF_cmdOff THEN StrSw.CmdOff := FALSE; END_IF;
  			ELSIF  StrSw.ISVALIDREF_cmdOff THEN StrSw.CmdOff := FALSE;  END_IF;
                                lastCmd := cmd;
  			errorCMDTimer(IN := false);
  			_commandErrorTimer := true;
  			StrSw.lastCmdIsOn := true;
  	(*cmd_close*) 2 :
  			IF StrSw.ISVALIDREF_cmdOff THEN StrSw.CmdOff := TRUE;
  				IF StrSw.ISVALIDREF_cmdOn THEN StrSw.CmdOn := FALSE; END_IF;
  			ELSIF StrSw.ISVALIDREF_cmdOn THEN StrSw.CmdOn := FALSE; END_IF;
                                lastCmd := cmd;
  			errorCMDTimer(IN := false);
  			_commandErrorTimer := true;
  			StrSw.lastCmdIsOn := false;
  	(*cmd_reset*) 3 :    IF StrSw.ISVALIDREF_statOn OR StrSw.ISVALIDREF_statOff THEN
  			StrSw.CmdOn := FALSE;
  			StrSw.CmdOff := FALSE;
                                lastCmd :=0;
  			_commandErrorTimer := false;
  			StrSw.lastCmdIsOn := false;
                                 END_IF;
  	END_CASE;
  	source_for_Status := source;
  	cmd_for_Status := cmd;
  	command_error_for_Status := 0;
  END_IF;

  errorCMDTimer(In := _commandErrorTimer, PT :=T#10s);

  (* ---- алгоритм  для команды ВКЛючить ---- *)
  IF (StrSw.onStatus = _statusDualInput.STATUS_ON) and StrSw.lastCmdIsOn then
  	IF StrSw.ISVALIDREF_cmdOn AND StrSw.ISVALIDREF_cmdOff then  StrSw.cmdOn := false; END_IF;

  	 errorCMDTimer(In := false);
  	 _commandErrorTimer := false;
  	 cmd_for_Status := 0;
  	 source_for_Status := 0;
  END_IF;

  (* ---- off ---- *)
  IF (StrSw.onStatus = _statusDualInput.STATUS_OFF) and (NOT StrSw.lastCmdIsOn) then
  	IF StrSw.ISVALIDREF_cmdOn AND StrSw.ISVALIDREF_cmdOff then  StrSw.cmdOff := false; END_IF;

  	 errorCMDTimer(In := false);
  	 _commandErrorTimer := false;
  	 cmd_for_Status := 0;
  	 source_for_Status := 0;
  END_IF;

  (* ---- ошибка исполнения команды ---- *)
  if errorCMDTimer.Q and (cmd_for_Status <> 0) then
  	command_error_for_Status :=  cmd_for_Status;
  	_commandErrorTimer := false;
  	StrSw.CmdOn := false;
  	StrSw.CmdOff := false;
  	lastCmd := 0;
  end_if;

  (* ---- сброс ошибки команды ---- *)
  StrSw.CommandFault := command_error_for_Status <> 0;
  _errorReset(IN := command_error_for_Status <> 0, PT := T#5S);
  IF _errorReset.Q THEN
  	cmd_for_Status := 0;
  	source_for_Status := 0;
  	command_error_for_Status := 0;
  END_IF;

  outputsSets(in := (StrSw.ISVALIDREF_cmdOn and StrSw.cmdOn ) OR (StrSw.ISVALIDREF_cmdOff and StrSw.cmdOff), PT := T#2S);
  	IF NOT outputsSets.Q THEN
  		StrSw.BreakCmdOn := inBreakCmdOn._inversed AND
                      inBreakCmdOn.reliability AND StrSw.ISVALIDREF_inBreakCmdOn;

  		StrSw.BreakCmdOff := inBreakCmdOff._inversed
                      AND inBreakCmdOff.reliability AND StrSw.ISVALIDREF_inBreakCmdOff;
  	END_IF;

  cmdOn := StrSw.cmdOn;
  cmdOff:= StrSw.cmdOff;

  (* ---- формирование зашифрованного статуса для АРМа ---- *)
  StrSw.status := shl(BYTE_TO_DWORD(source_for_Status), 29)
  		OR shl(BYTE_TO_DWORD(cmd_for_Status), 26)
  		OR shl(BYTE_TO_DWORD(command_error_for_Status), 23)
  		OR shl(bool_to_DWORD(StrSw.sdvig), 22)
  		OR shl(bool_to_DWORD(StrSw.OpcCommandsDisabled), 21)
                      OR shl(bool_to_DWORD(StrSw.lastCmdIsOn), 14)
                      OR shl(BOOL_TO_DWORD(StrSw.BreakCmdOff), 13)
  		OR shl(BOOL_TO_DWORD(StrSw.BreakCmdOn), 12)
  		OR shl(BOOL_TO_DWORD(StrSw.ErrorBlock), 11)
  		OR shl(BOOL_TO_DWORD(StrSw.ErrorPowerOff), 10)
  		OR shl(BOOL_TO_DWORD(StrSw.Manual), 8)
  		OR shl(BOOL_TO_DWORD(StrSw.Auto), 7)
  		OR shl(BOOL_TO_DWORD(StrSw.Distance), 6)
  		OR shl(BOOL_TO_DWORD(StrSw.Local), 5)
  		OR shl(BOOL_TO_DWORD(StrSw.Ns), 4)
                  	OR shl(BOOL_TO_DWORD(StrSw.Accident ),3)
  		OR BYTE_TO_DWORD(StrSw.onStatus);
END_FUNCTION_BLOCK

FUNCTION_BLOCK fb_AiProtection_Init
  VAR_INPUT
    data_Ini : BOOL;
    controlLimit : BYTE;
    delay : TIME;
    inTag : BYTE;
    inRunOnStart : BOOL;
  END_VAR
  VAR_IN_OUT
    str_AIp : struct_AiProtection;
  END_VAR
  VAR_OUTPUT
    Init : BOOL    := FALSE;
  END_VAR

  (*****            Функциональный блок переинициализации структуры  AiProtection          *****)

   Init := FALSE;

      IF data_Ini THEN                            (* Параметрам требуется переинициализация. *)
          str_AIp.controlLimit        := controlLimit;
          str_AIp.delay               := delay;
          str_AIp.inTag               := inTag;
          str_AIp.inRunOnStart        := inRunOnStart;

          data_Ini:=FALSE;
          Init := TRUE;
      END_IF;
      IF Init THEN
          controlLimit:= 0;
          delay:= T#0S;
          inTag:= 0;
          inRunOnStart:= FALSE;
      END_IF;
END_FUNCTION_BLOCK

FUNCTION_BLOCK fb_Switch_Init
  VAR_INPUT
    data_Ini : BOOL;
    ISVALIDREF_statOn : BOOL;
    ISVALIDREF_statOff : BOOL;
    ISVALIDREF_cmdOn : BOOL;
    ISVALIDREF_cmdOff : BOOL;
    ISVALIDREF_inBreakCmdOn : BOOL;
    ISVALIDREF_inBreakCmdOff : BOOL;
  END_VAR
  VAR_IN_OUT
    str_Sw : struct_Switch;
  END_VAR
  VAR_OUTPUT
    Init : BOOL    := FALSE;
  END_VAR

  (*****            Функциональный блок переинициализации структуры  Switch          *****)

   Init := FALSE;

      IF data_Ini THEN                            (* Параметрам требуется переинициализация. *)
          str_Sw.ISVALIDREF_statOn                := ISVALIDREF_statOn;
          str_Sw.ISVALIDREF_statOff               := ISVALIDREF_statOff;
          str_Sw.ISVALIDREF_cmdOn                 := ISVALIDREF_cmdOn;
          str_Sw.ISVALIDREF_cmdOff                := ISVALIDREF_cmdOff;
          str_Sw.ISVALIDREF_inBreakCmdOn          := ISVALIDREF_inBreakCmdOn;
          str_Sw.ISVALIDREF_inBreakCmdOff         := ISVALIDREF_inBreakCmdOff;
          data_Ini:=FALSE;
          Init := TRUE;
      END_IF;
  IF Init THEN
          ISVALIDREF_statOn:= FALSE;
          ISVALIDREF_statOff:= FALSE;
          ISVALIDREF_cmdOn:= FALSE;
          ISVALIDREF_cmdOff:= FALSE;
          ISVALIDREF_inBreakCmdOn:= FALSE;
          ISVALIDREF_inBreakCmdOff:= FALSE;
  END_IF;
END_FUNCTION_BLOCK

FUNCTION_BLOCK fb_DiProtection_Init
  VAR_INPUT
    data_Ini : BOOL;
    delay : TIME;
    inTag : BYTE;
    inRunOnStart : BOOL;
  END_VAR
  VAR_IN_OUT
    str_DIp : struct_DiProtection;
  END_VAR
  VAR_OUTPUT
    Init : BOOL    := FALSE;
  END_VAR

  (*****            Функциональный блок переинициализации структуры  AiProtection          *****)

   Init := FALSE;

      IF data_Ini THEN                            (* Параметрам требуется переинициализация. *)
          str_DIp.delay               := delay;
          str_DIp.inTag               := inTag;
          str_DIp.inRunOnStart        := inRunOnStart;

          data_Ini:=FALSE;
          Init := TRUE;
      END_IF;
      IF Init THEN
          delay:= T#0S;
          inTag:= 0;
          inRunOnStart:= FALSE;
      END_IF;
END_FUNCTION_BLOCK

FUNCTION_BLOCK fb_AiProtection
  VAR_INPUT
    ai : struct_AI;
  END_VAR
  VAR_IN_OUT
    StrAIp : struct_AiProtection;
  END_VAR
  VAR
    _sunpackerCommand : fb_sunpackerCommand;
    _signalingTp : TOF;
    _statusAi : TYPE_StatusAi;
    source : BYTE;
    cmd : BYTE;
    lastCmd : BYTE;
    source_for_Status : BYTE;
    cmd_for_Status : BYTE;
    command_error_for_Status : BYTE;
    resetCmdTimer : TON;
    resetCmdTimerPriznak : BOOL;
    signalinTimer : TON;
    timer : TON;
    SignalingTrig : R_TRIG;
    SignalingFTrig : F_TRIG;
    SignalingAi : BOOL;
  END_VAR

  timer(IN :=(ai.interval=StrAIp.controlLimit) AND (ai.interval >= _statusAi.normal) AND StrAIp.isRunning, PT :=StrAIp.delay);
  SignalingTrig(CLK := timer.Q);
  IF SignalingTrig.Q THEN
  	SignalingAi := TRUE;
  END_IF;
  SignalingFTrig(CLK := timer.Q);
  IF SignalingFTrig.Q THEN
  	SignalingAi := FALSE;
  END_IF;

  StrAIp.Tag := StrAIp.inTag;
  StrAIp.RunOnStart := StrAIp.inRunOnStart;

  StrAIp.CanRun := StrAIp.inCanRun;

  StrAIp.OpcCommandsDisabled := StrAIp.inOpcCommandsDisabled;

  (* ---- Если управление с ВУ заблокировано, то передаем команду из алгоритма ---- *)
  IF StrAIp.inOpcCommandsDisabled THEN
  	StrAIp.inCommand := StrAIp.inCommand_Alg;
  ELSE (* иначе передаем команду с АРМа*)
  	StrAIp.inCommand := StrAIp.inCommand_ARM;
  END_IF;

  _sunpackerCommand(command := StrAIp.inCommand);
  	source := _sunpackerCommand.source;
  	cmd := _sunpackerCommand.cmd;

  IF cmd <> 0 AND lastCmd <> cmd AND (((NOT StrAIp.opcCommandsDisabled) AND source > 0) OR source = 0) then

  	CASE BYTE_TO_INT(cmd) OF
  		(*cmdRun*) 1: 	IF        NOT StrAIp.Remont THEN
  					StrAIp.isEnded := FALSE;
  					StrAIp.hasError 	:= FALSE;
  					StrAIp.isRunning := TRUE;

  					cmd_for_Status := cmd;
  					source_for_Status := source;
  					command_error_for_Status := 0;
  				ELSE
  					StrAIp.isRunning := FALSE;
  					StrAIp.isEnded := FALSE;
  					StrAIp.hasError 	:= FALSE;

  					cmd_for_Status := 0;
  					source_for_Status := source;
  					command_error_for_Status := cmd;
  				END_IF;
                                          StrAIp.inopcCommandsDisabled:=FALSE;

  		(*cmdReset*) 2: 	StrAIp.isRunning := FALSE;
  				StrAIp.isEnded := FALSE;
  				StrAIp.hasError 	:= FALSE;
  				SignalingAi := FALSE;
  				StrAIp.Check := FALSE;
                                          (*StrAIp.Remont := FALSE;*)
  				cmd_for_Status := cmd;
  				source_for_Status := source;
  				command_error_for_Status := 0;
                                          StrAIp.inopcCommandsDisabled:=FALSE;

  	(*cmd_setRemont*) 4 :	StrAIp.Remont := TRUE;
  				(*StrAIp.isRunning := FALSE;*)

  				cmd_for_Status := cmd;
  				source_for_Status := source;
  				command_error_for_Status := 0;
  	(*cmd_resetRemont*) 5 : 	(*IF (ai.interval=StrAIp.controlLimit) THEN
  					cmd_for_Status := 0;
  					source_for_Status := 0;
  					command_error_for_Status := cmd;
  				ELSE*)
  					StrAIp.Remont := FALSE;
  					(*StrAIp.isRunning := TRUE;*)

  					cmd_for_Status := cmd;
  					source_for_Status := source;
  					command_error_for_Status := 0;
  				(*END_IF;*)
  	(*cmd_setCheck*) 6 : 	StrAIp.Check := TRUE;

  				cmd_for_Status := cmd;
  				source_for_Status := source;
  				command_error_for_Status := 0;
  	END_CASE;
  	resetCmdTimer(IN := false);
  	resetCmdTimerPriznak := TRUE;
  END_IF;
  lastCmd := cmd;

  resetCmdTimer(IN := resetCmdTimerPriznak);
  IF resetCmdTimer.Q THEN
  	resetCmdTimerPriznak := FALSE;
  	source_for_Status := 0;
  	cmd_for_Status := 0;
  	command_error_for_Status := 0;
  END_IF;

  IF StrAIp.isRunning AND NOT StrAIp.Remont AND NOT StrAIp.Check THEN
  	StrAIp.Signaling := SignalingAi;
  	StrAIp.SignalingTP := _signalingTp.Q;
  ELSE
  	StrAIp.Signaling := 0;
  	StrAIp.SignalingTP := 0;
  END_IF;

  _signalingTp(in := StrAIp.Signaling, PT := T#1s);

  StrAIp.status :=  SHL(BYTE_TO_DWORD(source_for_Status), 29)
  			OR SHL(BYTE_TO_DWORD(cmd_for_Status), 26)
  			OR SHL(BYTE_TO_DWORD(command_error_for_Status), 23)
  			OR SHL(BOOL_TO_DWORD(StrAIp.OpcCommandsDisabled ), 21)
  			OR SHL(BOOL_TO_DWORD(StrAIp.Signaling), 16)
  			OR SHL(BOOL_TO_DWORD(StrAIp.RunOnStart ), 15)
  			OR SHL(BOOL_TO_DWORD(StrAIp.remont), 6)
  			OR SHL(BOOL_TO_DWORD(StrAIp.Check), 5)
  			OR SHL(BOOL_TO_DWORD(StrAIp.hasError), 4)
  			OR SHL(BOOL_TO_DWORD(StrAIp.SignalingTP), 3)
  			OR SHL(BOOL_TO_DWORD(StrAIp.CanRun), 2)
  			OR SHL(BOOL_TO_DWORD(StrAIp.isEnded), 1)
  			OR BOOL_TO_DWORD(StrAIp.isRunning);
END_FUNCTION_BLOCK

FUNCTION_BLOCK fb_DiProtection
  VAR_INPUT
    di : struct_singleSignal;
  END_VAR
  VAR_IN_OUT
    StrDIp : struct_DiProtection;
  END_VAR
  VAR
    _sunpackerCommand : fb_sunpackerCommand;
    _ProtectionTags : TYPE_ProtectionTags;
    _signalingTp : TOF;
    timer : TON;
    SignalingTrig : R_TRIG;
    SignalingFTrig : F_TRIG;
    SignalingDi : BOOL;
    source : BYTE;
    cmd : BYTE;
    lastCmd : BYTE;
    source_for_Status : BYTE;
    cmd_for_Status : BYTE;
    command_error_for_Status : BYTE;
    resetCmdTimer : TON;
    resetCmdTimerPriznak : BOOL;
    signalinTimer : TON;
    runOnStart_Trig : R_TRIG;
  END_VAR

  timer(IN := di.Q AND StrDIp.isRunning  , PT := StrDIp.delay);
  SignalingTrig(CLK := timer.Q);
  IF SignalingTrig.Q THEN
  	SignalingDi := TRUE;
  END_IF;
  SignalingFTrig(CLK := timer.Q);
  IF SignalingFTrig.Q THEN
  	SignalingDi := FALSE;
  END_IF;

  StrDIp.Tag := StrDIp.inTag;
  StrDIp.RunOnStart := StrDIp.inRunOnStart;

  StrDIp.CanRun := StrDIp.inCanRun;

  StrDIp.OpcCommandsDisabled := StrDIp.inOpcCommandsDisabled;

  (* ---- Если управление с ВУ заблокировано, то передаем команду из алгоритма ---- *)
  IF StrDIp.inOpcCommandsDisabled THEN
  	StrDIp.inCommand := StrDIp.inCommand_Alg;
  ELSE (* иначе передаем команду с АРМа*)
  	StrDIp.inCommand := StrDIp.inCommand_ARM;
  END_IF;

  _sunpackerCommand(command := StrDIp.inCommand);
  	source := _sunpackerCommand.source;
  	cmd := _sunpackerCommand.cmd;

  IF cmd <> 0 AND lastCmd <> cmd AND (((NOT StrDIp.opcCommandsDisabled) AND source > 0) OR source = 0) then

  	CASE BYTE_TO_INT(cmd) OF
  	        (*cmdRun*) 1: 	IF        NOT StrDIp.Remont THEN
  					StrDIp.isEnded := FALSE;
  					StrDIp.hasError 	:= FALSE;
  					StrDIp.isRunning := TRUE;
  					cmd_for_Status := cmd;
  					source_for_Status := source;
  					command_error_for_Status := 0;
  				ELSE
  					StrDIp.isRunning := FALSE;
  					StrDIp.isEnded := FALSE;
  					StrDIp.hasError 	:= FALSE;

  					cmd_for_Status := 0;
  					source_for_Status := source;
  					command_error_for_Status := cmd;
  				END_IF;
                                          StrDIp.inOpcCommandsDisabled:=FALSE;

                  (*cmdReset*) 2: 	StrDIp.isRunning := FALSE;
  				StrDIp.isEnded := FALSE;
  				StrDIp.hasError 	:= FALSE;
  				SignalingDi:= FALSE;
  				StrDIp.Check := FALSE;
  				cmd_for_Status := cmd;
  				source_for_Status := source;
  				command_error_for_Status := 0;
                                         StrDIp.inOpcCommandsDisabled:=FALSE;

  	(*cmd_setRemont*) 4 :	StrDIp.Remont := TRUE;
  				(*StrDIp.isRunning := FALSE;*)

  				cmd_for_Status := cmd;
  				source_for_Status := source;
  				command_error_for_Status := 0;
          (*cmd_resetRemont*) 5 : 	(*IF di.Q THEN
  					cmd_for_Status := 0;
  					source_for_Status := 0;
  					command_error_for_Status := cmd;
  				ELSE*)
  					StrDIp.Remont := FALSE;
  					(*StrDIp.isRunning := TRUE;*)

  					cmd_for_Status := cmd;
  					source_for_Status := source;
  					command_error_for_Status := 0;
  				(*END_IF;*)
  	(*cmd_setCheck*) 6 : 	StrDIp.Check := TRUE;

  				cmd_for_Status := cmd;
  				source_for_Status := source;
  				command_error_for_Status := 0;
  	END_CASE;
  	resetCmdTimer(IN := false);
  	resetCmdTimerPriznak := TRUE;
  END_IF;
  lastCmd := cmd;

  resetCmdTimer(IN := resetCmdTimerPriznak);
  IF resetCmdTimer.Q THEN
  	resetCmdTimerPriznak := FALSE;
  	source_for_Status := 0;
  	cmd_for_Status := 0;
  	command_error_for_Status := 0;
  END_IF;

  IF StrDIp.isRunning AND NOT StrDIp.Remont AND NOT StrDIp.Check THEN
  	StrDIp.Signaling := SignalingDi;
  	StrDIp.SignalingTP := _signalingTp.Q;
  ELSE
  	StrDIp.Signaling := 0;
  	StrDIp.SignalingTP := 0;
  END_IF;

  _signalingTp(in := StrDIp.Signaling, PT := T#1s);

  StrDIp.status :=  SHL(BYTE_TO_DWORD(source_for_Status), 29)
  			OR SHL(BYTE_TO_DWORD(cmd_for_Status), 26)
  			OR SHL(BYTE_TO_DWORD(command_error_for_Status), 23)
  			OR SHL(BOOL_TO_DWORD(StrDIp.OpcCommandsDisabled ), 21)
  			OR SHL(BOOL_TO_DWORD(StrDIp.Signaling), 16)
  			OR SHL(BOOL_TO_DWORD(StrDIp.RunOnStart ), 15)
  			OR SHL(BOOL_TO_DWORD(StrDIp.remont), 6)
  			OR SHL(BOOL_TO_DWORD(StrDIp.Check), 5)
  			OR SHL(BOOL_TO_DWORD(StrDIp.hasError), 4)
  			OR SHL(BOOL_TO_DWORD(StrDIp.SignalingTP), 3)
  			OR SHL(BOOL_TO_DWORD(StrDIp.CanRun), 2)
  			OR SHL(BOOL_TO_DWORD(StrDIp.isEnded), 1)
  			OR BOOL_TO_DWORD(StrDIp.isRunning);
END_FUNCTION_BLOCK

FUNCTION_BLOCK Proc_Protection
  VAR_EXTERNAL
    Protections : ProtectionsConfig;
    Ai : AiConfig;
    Im : ImConfig;
  END_VAR
  VAR
    fb_Ap1 : fb_AiProtection;
    fb_AiP1 : fb_AiProtection;
    fb_AiP2 : fb_AiProtection;
    fb_AiP3 : fb_AiProtection;
    fb_DiP1 : fb_DiProtection;
    fb_DiP2 : fb_DiProtection;
    fb_DiP3 : fb_DiProtection;
    fb_DiP4 : fb_DiProtection;
    fb_DiP5 : fb_DiProtection;
  END_VAR

  fb_Ap1(ai := Ai.A1, StrAIp := Protections.Ap1);

  fb_AiP1(ai := Ai.A2, StrAIp := Protections.AiP1);

  fb_AiP2(ai := Ai.A1, StrAIp := Protections.AiP2);

  fb_AiP3(ai := Ai.A2, StrAIp := Protections.AiP3);

  fb_DiP1(di := Im.SingleSignals.SI2, StrDIp := Protections.DiP1);

  fb_DiP2(di := Im.SingleSignals.SI0, StrDIp := Protections.DiP2);

  fb_DiP3(di := Im.SingleSignals.SI0, StrDIp := Protections.DiP3);

  fb_DiP4(di := Im.SingleSignals.SI2, StrDIp := Protections.DiP4);

  fb_DiP5(di := Im.SingleSignals.SI4, StrDIp := Protections.DiP5);
END_FUNCTION_BLOCK

FUNCTION_BLOCK fb_Kran_Init
  VAR_INPUT
    data_Ini : BOOL;
    ISVALIDREF_statOn : BOOL;
    ISVALIDREF_statOff : BOOL;
    ISVALIDREF_cmdOn : BOOL;
    ISVALIDREF_cmdOff : BOOL;
    ISVALIDREF_inSo : BOOL;
    ISVALIDREF_inSz : BOOL;
    ISVALIDREF_inDp : BOOL    := False;
    continueHoldCommand : TIME;
  END_VAR
  VAR_IN_OUT
    str_Kr : struct_Kran;
  END_VAR
  VAR_OUTPUT
    Init : BOOL    := FALSE;
  END_VAR

  (*****            Функциональный блок переинициализации структуры  Kran          *****)

          Init := False;

      IF data_Ini THEN                            (* Параметрам требуется переинициализация. *)
          str_Kr.ISVALIDREF_statOn                := ISVALIDREF_statOn;
          str_Kr.ISVALIDREF_statOff               := ISVALIDREF_statOff;
          str_Kr.ISVALIDREF_cmdOn                 := ISVALIDREF_cmdOn;
          str_Kr.ISVALIDREF_cmdOff                := ISVALIDREF_cmdOff;
          str_Kr.ISVALIDREF_inSo                  := ISVALIDREF_inSo;
          str_Kr.ISVALIDREF_inSz                  := ISVALIDREF_inSz;
          str_Kr.ISVALIDREF_inDp                  := ISVALIDREF_inDp;
          str_Kr.continueHoldCommand              := continueHoldCommand;

          data_Ini:=False;
          Init := TRUE;
     END_IF;
   IF Init THEN
          ISVALIDREF_statOn:= false;
          ISVALIDREF_statOff:= false;
          ISVALIDREF_cmdOn:= false;
          ISVALIDREF_cmdOff:= false;
          ISVALIDREF_inSo:= false;
          ISVALIDREF_inSz:= false;
          ISVALIDREF_inDp:= false;
          continueHoldCommand:= T#0S;
    END_IF;
END_FUNCTION_BLOCK

FUNCTION_BLOCK fb_OilPump_Init
  VAR_INPUT
    data_Ini : BOOL;
    ISVALIDREF_statOn : BOOL;
    ISVALIDREF_statOff : BOOL;
    ISVALIDREF_cmdOn : BOOL;
    ISVALIDREF_cmdOff : BOOL;
    ISVALIDREF_inBreakCmdOn : BOOL;
    ISVALIDREF_inBreakCmdOff : BOOL;
  END_VAR
  VAR_IN_OUT
    str_Op : struct_OilPump;
  END_VAR
  VAR_OUTPUT
    Init : BOOL    := FALSE;
  END_VAR

  (*****            Функциональный блок переинициализации структуры  НУ          *****)

   Init := FALSE;

      IF data_Ini THEN                            (* Параметрам требуется переинициализация. *)
          str_Op.ISVALIDREF_statOn                := ISVALIDREF_statOn;
          str_Op.ISVALIDREF_statOff               := ISVALIDREF_statOff;
          str_Op.ISVALIDREF_cmdOn                 := ISVALIDREF_cmdOn;
          str_Op.ISVALIDREF_cmdOff                := ISVALIDREF_cmdOff;
          str_Op.ISVALIDREF_inBreakCmdOn          := ISVALIDREF_inBreakCmdOn;
          str_Op.ISVALIDREF_inBreakCmdOff         := ISVALIDREF_inBreakCmdOff;
          data_Ini:=FALSE;
          Init := TRUE;
      END_IF;

          ISVALIDREF_statOn:= FALSE;
          ISVALIDREF_statOff:= FALSE;
          ISVALIDREF_cmdOn:= FALSE;
          ISVALIDREF_cmdOff:= FALSE;
          ISVALIDREF_inBreakCmdOn:= FALSE;
          ISVALIDREF_inBreakCmdOff:= FALSE;
END_FUNCTION_BLOCK

FUNCTION_BLOCK fb_SectionSwitch_Init
  VAR_INPUT
    data_Ini : BOOL;
    ISVALIDREF_statOn : BOOL;
    ISVALIDREF_statOff : BOOL;
    ISVALIDREF_cmdOn : BOOL;
    ISVALIDREF_cmdOff : BOOL;
    ISVALIDREF_inBreakCmdOn : BOOL;
    ISVALIDREF_inBreakCmdOff : BOOL;
    ISVALIDREF_basketRolledIn : BOOL;
    ISVALIDREF_basketRolledOut : BOOL;
    ISVALIDREF_basketTest : BOOL;
  END_VAR
  VAR_IN_OUT
    str_Sw : struct_SectionSwitch;
  END_VAR
  VAR_OUTPUT
    Init : BOOL    := FALSE;
  END_VAR

  (*****            Функциональный блок переинициализации структуры  МВ          *****)

   Init := FALSE;

      IF data_Ini THEN                            (* Параметрам требуется переинициализация. *)
          str_Sw.ISVALIDREF_statOn                := ISVALIDREF_statOn;
          str_Sw.ISVALIDREF_statOff               := ISVALIDREF_statOff;
          str_Sw.ISVALIDREF_cmdOn                 := ISVALIDREF_cmdOn;
          str_Sw.ISVALIDREF_cmdOff                := ISVALIDREF_cmdOff;
          str_Sw.ISVALIDREF_inBreakCmdOn          := ISVALIDREF_inBreakCmdOn;
          str_Sw.ISVALIDREF_inBreakCmdOff         := ISVALIDREF_inBreakCmdOff;
          str_Sw.ISVALIDREF_basketRolledIn        := ISVALIDREF_basketRolledIn;
          str_Sw.ISVALIDREF_basketRolledOut       := ISVALIDREF_basketRolledOut;
          str_Sw.ISVALIDREF_basketTest            := ISVALIDREF_basketTest;
          data_Ini:=FALSE;
          Init := TRUE;
      END_IF;
  IF Init THEN
          ISVALIDREF_statOn:= FALSE;
          ISVALIDREF_statOff:= FALSE;
          ISVALIDREF_cmdOn:= FALSE;
          ISVALIDREF_cmdOff:= FALSE;
          ISVALIDREF_inBreakCmdOn:= FALSE;
          ISVALIDREF_inBreakCmdOff:= FALSE;
          ISVALIDREF_basketRolledIn:= FALSE;
          ISVALIDREF_basketRolledOut:= FALSE;
          ISVALIDREF_basketTest:= FALSE;
  END_IF;
END_FUNCTION_BLOCK

FUNCTION_BLOCK fb_singleSignal_Init
  VAR_INPUT
    data_Ini : BOOL;
    inverse : BOOL;
    DelayOn : TIME;
    DelayOff : TIME;
  END_VAR
  VAR_IN_OUT
    str_SS : struct_singleSignal;
  END_VAR
  VAR_OUTPUT
    Init : BOOL    := FALSE;
  END_VAR

  (*****            Функциональный блок переинициализации структуры  singleSignal          *****)
  Init := FALSE;

      IF data_Ini THEN                            (* Параметрам требуется переинициализация. *)
          str_SS.inverse                := inverse;
          str_SS.DelayOn                := DelayOn;
          str_SS.DelayOff               := DelayOff;

          data_Ini:=FALSE;
          Init := TRUE;
      END_IF;
   IF Init THEN
          inverse := FALSE;
          DelayOn := T#0S;
          DelayOff:= T#0S;
   END_IF;
END_FUNCTION_BLOCK

FUNCTION_BLOCK fb_singleOutput_Init
  VAR_INPUT
    data_Ini : BOOL;
    inOpcCommandsDisabled : BOOL;
    wait_time : TIME;
  END_VAR
  VAR_IN_OUT
    str_SO : struct_singleOutput;
  END_VAR
  VAR_OUTPUT
    Init : BOOL    := FALSE;
  END_VAR

  (*****            Функциональный блок переинициализации структуры  singleOutput          *****)

  Init := FALSE;

      IF data_Ini THEN                            (* Параметрам требуется переинициализация. *)
          str_SO.inOpcCommandsDisabled    := inOpcCommandsDisabled;
          str_SO.wait_time                := wait_time;

           data_Ini:=FALSE;
          Init := TRUE;
      END_IF;
   IF Init THEN
          inOpcCommandsDisabled := FALSE;
          wait_time := T#0S;
     END_IF;
END_FUNCTION_BLOCK

FUNCTION_BLOCK Proc_Im_Init
  VAR_INPUT
    init : BOOL;
  END_VAR
  VAR
    stKr_Ini : fb_Kran_Init;
    stSw_Ini : fb_Switch_Init;
    stOp_Ini : fb_OilPump_Init;
    stSSw_Ini : fb_SectionSwitch_Init;
    stSs_Ini : fb_singleSignal_Init;
    stSo_Ini : fb_singleOutput_Init;
    inits : UINT;
  END_VAR
  VAR_INPUT
    initiales : UINT;
  END_VAR
  VAR_EXTERNAL
    Im : ImConfig;
  END_VAR

  stKr_Ini(str_Kr := Im.Kran1,
  ISVALIDREF_inDp := TRUE,
  ISVALIDREF_inSo := TRUE,
  ISVALIDREF_inSz := TRUE,
  ISVALIDREF_statOn := TRUE,
  ISVALIDREF_statOff := TRUE,
  ISVALIDREF_cmdOn := TRUE,
  ISVALIDREF_cmdOff := TRUE);
  inits := inits + BOOL_TO_UINT(stKr_Ini.Init);

  stKr_Ini(str_Kr := Im.Kran4,
  ISVALIDREF_inDp := TRUE,
  ISVALIDREF_inSo := TRUE,
  ISVALIDREF_inSz := TRUE,
  ISVALIDREF_statOn := TRUE,
  ISVALIDREF_statOff := TRUE,
  ISVALIDREF_cmdOn := TRUE,
  ISVALIDREF_cmdOff := TRUE);
  inits := inits + BOOL_TO_UINT(stKr_Ini.Init);

  stKr_Ini(str_Kr := Im.Kran2,
  ISVALIDREF_inDp := TRUE,
  ISVALIDREF_inSo := TRUE,
  ISVALIDREF_inSz := TRUE,
  ISVALIDREF_statOn := TRUE,
  ISVALIDREF_statOff := TRUE,
  ISVALIDREF_cmdOn := TRUE,
  ISVALIDREF_cmdOff := TRUE);
  inits := inits + BOOL_TO_UINT(stKr_Ini.Init);

  stKr_Ini(str_Kr := Im.Kran3,
  ISVALIDREF_inDp := TRUE,
  ISVALIDREF_inSo := TRUE,
  ISVALIDREF_inSz := TRUE,
  ISVALIDREF_statOn := TRUE,
  ISVALIDREF_statOff := TRUE,
  ISVALIDREF_cmdOn := TRUE,
  ISVALIDREF_cmdOff := TRUE);
  inits := inits + BOOL_TO_UINT(stKr_Ini.Init);

  stOp_Ini(str_Op := Im.Nu,
  ISVALIDREF_inBreakCmdOn := TRUE,
  ISVALIDREF_inBreakCmdOff := TRUE,
  ISVALIDREF_statOn := TRUE,
  ISVALIDREF_statOff := TRUE,
  ISVALIDREF_cmdOn := TRUE,
  ISVALIDREF_cmdOff := TRUE);
  inits := inits + BOOL_TO_UINT(stOp_Ini.Init);

  stOp_Ini(str_Op := Im.Nu2,
  ISVALIDREF_inBreakCmdOn := TRUE,
  ISVALIDREF_inBreakCmdOff := TRUE,
  ISVALIDREF_statOn := TRUE,
  ISVALIDREF_statOff := TRUE,
  ISVALIDREF_cmdOn := TRUE,
  ISVALIDREF_cmdOff := TRUE);
  inits := inits + BOOL_TO_UINT(stOp_Ini.Init);

  stSSw_Ini(str_Sw := Im.Mv,
  ISVALIDREF_inBreakCmdOn := TRUE,
  ISVALIDREF_inBreakCmdOff := TRUE,
  ISVALIDREF_basketRolledIn := TRUE,
  ISVALIDREF_basketRolledout := TRUE,
  ISVALIDREF_basketTest := TRUE,
  ISVALIDREF_statOn := TRUE,
  ISVALIDREF_statOff := TRUE,
  ISVALIDREF_cmdOn := TRUE,
  ISVALIDREF_cmdOff := TRUE);
  inits := inits + BOOL_TO_UINT(stSSw_Ini.Init);

  stSSw_Ini(str_Sw := Im.SectionSwitch1);
  inits := inits + BOOL_TO_UINT(stSSw_Ini.Init);

  stSw_Ini(str_Sw := Im.Avom1,
  ISVALIDREF_inBreakCmdOn := TRUE,
  ISVALIDREF_inBreakCmdOff := TRUE,
  ISVALIDREF_statOn := TRUE,
  ISVALIDREF_statOff := TRUE,
  ISVALIDREF_cmdOn := TRUE,
  ISVALIDREF_cmdOff := TRUE);
  inits := inits + BOOL_TO_UINT(stSw_Ini.Init);

  stSw_Ini(str_Sw := Im.Avom2,
  ISVALIDREF_inBreakCmdOn := TRUE,
  ISVALIDREF_inBreakCmdOff := TRUE,
  ISVALIDREF_statOn := TRUE,
  ISVALIDREF_statOff := TRUE,
  ISVALIDREF_cmdOn := TRUE,
  ISVALIDREF_cmdOff := TRUE);
  inits := inits + BOOL_TO_UINT(stSw_Ini.Init);

  stSw_Ini(str_Sw := Im.Avom3,
  ISVALIDREF_inBreakCmdOn := TRUE,
  ISVALIDREF_inBreakCmdOff := TRUE,
  ISVALIDREF_statOn := TRUE,
  ISVALIDREF_statOff := TRUE,
  ISVALIDREF_cmdOn := TRUE,
  ISVALIDREF_cmdOff := TRUE);
  inits := inits + BOOL_TO_UINT(stSw_Ini.Init);

  stSw_Ini(str_Sw := Im.Avom4,
  ISVALIDREF_inBreakCmdOn := TRUE,
  ISVALIDREF_inBreakCmdOff := TRUE,
  ISVALIDREF_statOn := TRUE,
  ISVALIDREF_statOff := TRUE,
  ISVALIDREF_cmdOn := TRUE,
  ISVALIDREF_cmdOff := TRUE);
  inits := inits + BOOL_TO_UINT(stSw_Ini.Init);

  stSs_Ini(data_Ini := TRUE, inverse := FALSE, str_SS := Im.SingleSignals.SI0);
  inits := inits + BOOL_TO_UINT(stSs_Ini.Init);

  stSs_Ini(data_Ini := TRUE, inverse := FALSE, str_SS := Im.SingleSignals.SI1);
  inits := inits + BOOL_TO_UINT(stSs_Ini.Init);

  stSs_Ini(data_Ini := TRUE, inverse := FALSE, str_SS := Im.SingleSignals.SI2);
  inits := inits + BOOL_TO_UINT(stSs_Ini.Init);

  stSs_Ini(data_Ini := TRUE, inverse := FALSE, str_SS := Im.SingleSignals.SI3);
  inits := inits + BOOL_TO_UINT(stSs_Ini.Init);

  stSs_Ini(data_Ini := TRUE, inverse := FALSE, str_SS := Im.SingleSignals.SI4);
  inits := inits + BOOL_TO_UINT(stSs_Ini.Init);

  stSs_Ini(data_Ini := TRUE, inverse := FALSE, str_SS := Im.SingleSignals.SI5);
  inits := inits + BOOL_TO_UINT(stSs_Ini.Init);

  stSs_Ini(data_Ini := TRUE, inverse := FALSE, str_SS := Im.SingleSignals.SI6);
  inits := inits + BOOL_TO_UINT(stSs_Ini.Init);

  stSo_Ini(data_Ini := TRUE, inOpcCommandsDisabled := FALSE, str_SO := Im.SingleOutputs.So0);
  inits := inits + BOOL_TO_UINT(stSo_Ini.Init);

  stSo_Ini(data_Ini := TRUE, inOpcCommandsDisabled := FALSE, str_SO := Im.SingleOutputs.So1);
  inits := inits + BOOL_TO_UINT(stSo_Ini.Init);

  stSo_Ini(data_Ini := TRUE, inOpcCommandsDisabled := FALSE, str_SO := Im.SingleOutputs.So2);
  inits := inits + BOOL_TO_UINT(stSo_Ini.Init);

  stSo_Ini(data_Ini := TRUE, inOpcCommandsDisabled := FALSE, str_SO := Im.SingleOutputs.So3);
  inits := inits + BOOL_TO_UINT(stSo_Ini.Init);

  stSo_Ini(data_Ini := TRUE, inOpcCommandsDisabled := FALSE, str_SO := Im.SingleOutputs.So4);
  inits := inits + BOOL_TO_UINT(stSo_Ini.Init);

  stSo_Ini(data_Ini := TRUE, inOpcCommandsDisabled := FALSE, str_SO := Im.SingleOutputs.So5);
  inits := inits + BOOL_TO_UINT(stSo_Ini.Init);

  stSo_Ini(data_Ini := TRUE, inOpcCommandsDisabled := FALSE, str_SO := Im.SingleOutputs.So6);
  inits := inits + BOOL_TO_UINT(stSo_Ini.Init);

  stSo_Ini(data_Ini := TRUE, inOpcCommandsDisabled := FALSE, str_SO := Im.SingleOutputs.So7);
  inits := inits + BOOL_TO_UINT(stSo_Ini.Init);

  initiales := 0;
  IF init THEN initiales := inits; END_IF;
END_FUNCTION_BLOCK

FUNCTION_BLOCK fb_AI_Init
  VAR_INPUT
    data_Ini : BOOL;
    dLL : LREAL;
    dHL : LREAL;
    dLA : LREAL;
    dHA : LREAL;
    dLW : LREAL;
    dHW : LREAL;
    ISVALIDREF_LA : BOOL    := False;
    ISVALIDREF_HA : BOOL    := False;
    ISVALIDREF_LW : BOOL    := False;
    ISVALIDREF_HW : BOOL    := False;
    delayLA : TIME    := T#0S;
    delayLW : TIME    := T#0S;
    delayHW : TIME    := T#0S;
    delayHA : TIME    := T#0S;
    inpLL : LREAL    := 4000.0;
    inpHL : LREAL    := 20000.0;
    CurrentShotCircuit : LREAL    := 21000.0;
    CurrentBreakCircuit : LREAL    := 3700.0;
    maxChangeSpeed : LREAL;
    maxChangeSpeedDown : LREAL;
    histeresis : LREAL;
    aperturFilter : LREAL;
    exponentialFilter : LREAL;
    rassoglasovanie : LREAL;
    inOpcCommandsDisabled : BOOL;
  END_VAR
  VAR_IN_OUT
    strAI : struct_AI;
  END_VAR
  VAR_OUTPUT
    Init : BOOL    := FALSE;
  END_VAR

  (*****            Функциональный блок переинициализации структуры-дескриптора канала аналогового ввода.            *****)
       Init := false;

      IF data_Ini THEN                            (* Параметрам требуется переинициализация. *)
          strAI.dLL                := dLL;
          strAI.dHL                := dHL;
          strAI.dLA                := dLA;
          strAI.dHA                := dHA;
          strAI.dLW                := dLW;
          strAI.dHW                := dHW;
          strAI.ISVALIDREF_LA      := ISVALIDREF_LA;
          strAI.ISVALIDREF_HA      := ISVALIDREF_HA;
          strAI.ISVALIDREF_LW      := ISVALIDREF_LW;
          strAI.ISVALIDREF_HW      := ISVALIDREF_HW;
          strAI.delayLA            := delayLA;
          strAI.delayLW            := delayLW;
          strAI.delayHW            := delayHW;
          strAI.delayHA            := delayHA;
          strAI.inpLL              := inpLL;
          strAI.inpHL              := inpHL;
          strAI.CurrentShotCircuit := CurrentShotCircuit;
          strAI.CurrentBreakCircuit:= CurrentBreakCircuit;
          strAI.maxChangeSpeed     := maxChangeSpeed;
          strAI.maxChangeSpeedDown := maxChangeSpeedDown;
          strAI.histeresis         := histeresis;
          strAI.aperturFilter      := aperturFilter;
          strAI.exponentialFilter  := exponentialFilter;
          strAI.rassoglasovanie    := rassoglasovanie;
          strAI.rassoglasovanie    := rassoglasovanie;

          data_Ini:=false;
          Init := TRUE;
       END_IF;
    IF Init THEN
          dLL:= 0.0;
          dHL:= 0.0;
          dLA:= 0.0;
          dHA:= 0.0;
          dLW:= 0.0;
          dHW:= 0.0;
          inpLL:= 4000.0;
          inpHL:= 20000.0;
          CurrentShotCircuit:= 21000.0;
          CurrentBreakCircuit:= 3700.0;
          ISVALIDREF_LA:= false;
          ISVALIDREF_HA:= false;
          ISVALIDREF_LW:= false;
          ISVALIDREF_HW:= false;
          delayLA:= T#0S;
          delayLW:= T#0S;
          delayHW:= T#0S;
          delayHA:= T#0S;
          maxChangeSpeed:= 0.0;
          maxChangeSpeedDown:= 0.0;
          histeresis:= 0.0;
          aperturFilter:= 0.0;
          exponentialFilter:= 0.0;
          rassoglasovanie:= 0.0;
        END_IF;
END_FUNCTION_BLOCK

FUNCTION_BLOCK Proc_Ai_Init
  VAR_INPUT
    init : BOOL;
  END_VAR
  VAR
    stAI_Ini : fb_AI_Init;
    inits : UINT;
  END_VAR
  VAR_INPUT
    initiales : UINT;
  END_VAR
  VAR_EXTERNAL
    Ai : AiConfig;
  END_VAR

  inits := 0;

  stAI_Ini(data_Ini := TRUE, dLL := 0.0, dHL := 100.0,
  ISVALIDREF_LW := TRUE, dLW := 20.0,
  ISVALIDREF_HW := TRUE, dHW := 80.0,
  ISVALIDREF_LA := TRUE, dLA := 10.0,
  ISVALIDREF_HA := TRUE, dHA := 90.0,
  strAI := Ai.A1);
  inits := inits + BOOL_TO_UINT(stAI_Ini.Init);

  stAI_Ini(data_Ini := TRUE, dLL := 0.0, dHL := 100.0,
  ISVALIDREF_LW := TRUE, dLW := 20.0,
  ISVALIDREF_HW := TRUE, dHW := 80.0,
  ISVALIDREF_LA := TRUE, dLA := 10.0,
  ISVALIDREF_HA := TRUE, dHA := 90.0,
  strAI := Ai.A2);
  inits := inits + BOOL_TO_UINT(stAI_Ini.Init);

  initiales := 0;
  IF init THEN initiales := inits; END_IF;
END_FUNCTION_BLOCK

FUNCTION_BLOCK fb_AiSourceMlp
  VAR_INPUT
    arAIN : TItemAIN;
    err_mod : TItemDIN;
  END_VAR
  VAR_IN_OUT
    strAI : struct_AI;
  END_VAR
  VAR
    _statusAi : TYPE_StatusAi;
    _commandAnalog : TYPE_CommandAnalog;
    _sunpackerCommand : fb_sunpackerCommand;
    _AnalogLimitFlags : TYPE_AnalogLimitFlags;
    notReliable : BOOL;
    _lastValue : LREAL;
    resetCmdTimer : TON;
    _LastValueTimer : TON;
    resetCmdTimerPriznak : BOOL;
    k : LREAL;
    b : LREAL;
    ap : LREAL;
    raznitsa : LREAL;
    rABS : LREAL;
    h : LREAL;
    mismatch : LREAL;
    parametr : BYTE;
    source : BYTE;
    cmd : BYTE;
    lastCmd : BYTE;
    source_for_Status : BYTE;
    cmd_for_Status : BYTE;
    command_error_for_Status : BYTE;
    onInit : BOOL;
    off_trig : R_TRIG;
    on_trig : R_TRIG;
    remont_trig : R_TRIG;
    LL_trig : R_TRIG;
    HL_trig : R_TRIG;
    Normal_trig : R_TRIG;
    Nedostover_trig : R_TRIG;
  END_VAR

  strAI.opcCommandsDisabled := strAI.inopcCommandsDisabled ;

  (* ---- При первом пуске принимаем значение уставок ---- *)
  IF NOT onInit THEN

            strAI.LL := strAI.dLL;
            strAI.HL := strAI.dHL;

            IF strAI.ISVALIDREF_HA THEN strAI.HA := strAI.dHA; END_IF;

            IF strAI.ISVALIDREF_LA THEN strAI.LA := strAI.dLA; END_IF;

            IF strAI.ISVALIDREF_HW THEN strAI.HW := strAI.dHW; END_IF;

            IF strAI.ISVALIDREF_LW THEN strAI.LW := strAI.dLW; END_IF;

  	onInit  := TRUE;
  END_IF;

  (* ---- пересчет тока в физ величину ---- *)
  k := (strAI.HL - strAI.LL)/(strAI.inpHl - strAI.inpLL);
  b := strAI.LL - k * strAI.inpLL;
  strAI.value := k * arAIN.dblValue + b;

  (* ---- определение обрыва и кз ----- *)

  strAI.blConnect :=(*(UINT_TO_WORD(arAIN.wFlags) = 1472) and*) (UINT_TO_WORD(err_mod.wValue) = 20) and (UINT_TO_WORD(err_mod.wFlags) = 192);
  IF NOT strAI.blConnect THEN
      strAI.interval := _statusAi.NOTDEFINED;
  ELSIF ((arAIN.dblValue < strAI.currentBreakCircuit) AND (strAI.currentBreakCircuit > 0.0)) OR ((strAI.interval = _statusAi.LL) AND (arAIN.dblValue < (strAI.currentBreakCircuit + 100.0))) THEN
      strAI.interval := _statusAi.LL;
  ELSIF ((arAIN.dblValue > strAI.currentShotCircuit) AND (strAI.currentShotCircuit > 0.0)) OR ((strAI.interval = _statusAi.HL) AND (arAIN.dblValue > (strAI.currentShotCircuit - 100.0))) THEN
      strAI.interval := _statusAi.HL;
  ELSE
      strAI.interval := _statusAi.normal;
  END_IF;

  IF NOT strAI.imit THEN
  	(* Расчет апертурного фильтра*)
  	ap := strAI.aperturFilter * 0.01 * (strAI.HL - strAI.LL);
  	IF strAI.aperturFilter <> 0.0 THEN raznitsa := strAI.value- _lastValue;
  		IF 	raznitsa < 0.0 	THEN 	rABS := -raznitsa; 		ELSE 	rABS := raznitsa; 		END_IF;
  		IF 	rABS > ap 	THEN 	strAI.value := strAI.value;	ELSE 	strAI.value := _lastValue; 	END_IF;
  	END_IF;

  	(* Расчет экпоненциального фильтра*)
  	IF strAI.exponentialFilter <> 0.0 THEN strAI.value := (strAI.exponentialFilter * strAI.value) + ((1.0 - strAI.exponentialFilter) * _lastValue); END_IF;
  ELSE
  	strAI.interval := _statusAi.normal;
  END_IF;

  IF notReliable THEN strAI.interval := _statusAi.NOTRELIABLE; END_IF;

  IF NOT notReliable THEN
  	IF strAI.interval >= _statusAi.normal THEN
  		strAI.interval := _statusAi.NOTDEFINED;
  		h := strAI.histeresis* 0.01 * (strAI.HL-strAI.LL);
  		(*определение выхода за аппаратные границы вынесено в GetData.здесь только для нужд имитации*)
  		IF strAI.imit THEN
  			mismatch := strAI.rassoglasovanie * 0.01 * (strAI.HL - strAI.LL);
  			IF ( strAI.value < strAI.LL - mismatch)   THEN strAI.interval := _statusAi.LL;
  			ELSIF  (strAI.value > strAI.Hl + mismatch) THEN strAI.interval := _statusAi.HL; END_IF;
  		ELSE
  			strAI.interval := _statusAi.normal;
  			IF strAI.ISVALIDREF_LA AND NOT strAI.Disabled_LA AND (strAI.interval = _statusAi.normal) THEN
  				IF (strAI.value  < strAI.LA) OR ((strAI.interval = _statusAi.LA)  AND ((strAI.value - h) < strAI.LA))  THEN
  					strAI.interval := _statusAi.LA;
  				END_IF;
  			END_IF;
  			IF strAI.ISVALIDREF_HA  AND NOT strAI.Disabled_HA AND (strAI.interval = _statusAi.normal)  THEN
  				IF (strAI.value > strAI.HA) OR ((strAI.interval = _statusAi.HA)  AND ((strAI.value + h) > strAI.HA))  THEN
  					strAI.interval := _statusAi.HA;
  				END_IF;
  			END_IF;
  			IF strAI.ISVALIDREF_LW AND NOT strAI.Disabled_LW AND (strAI.interval = _statusAi.normal)  THEN
  				IF (strAI.value < strAI.LW) OR ((strAI.interval = _statusAi.LW)  AND ((strAI.value - h) < strAI.LW)) THEN
  					strAI.interval := _statusAi.LW;
  				END_IF;
  			END_IF;
  			IF strAI.ISVALIDREF_HW AND NOT strAI.Disabled_HW  AND (strAI.interval = _statusAi.normal) THEN
  				IF (strAI.value > strAI.HW)  OR ((strAI.interval = _statusAi.HW)  AND ((strAI.value + h) > strAI.HW))   THEN
  					strAI.interval := _statusAi.HW;
  				END_IF;
  			END_IF;
  		END_IF;
  	END_IF;
  ELSE
  	strAI.interval := _statusAi.NOTRELIABLE;
  END_IF;

  IF strAI.remont THEN strAI.interval := _statusAi.NOTDEFINED; END_IF;

  (* ---- Если управление с ВУ заблокировано, то  передаем команду из алгоритма ---- *)
  IF strAI.inOpcCommandsDisabled THEN
  	strAI.inCommand := strAI.inCommand_Alg;
  ELSE (* иначе передаем команду с АРМа*)
  	strAI.inCommand := strAI.inCommand_ARM;
  END_IF;

  _sunpackerCommand(command := strAI.inCommand);
  	source := _sunpackerCommand.source;
  	parametr := _sunpackerCommand.parametr;
  	cmd := _sunpackerCommand.cmd;

  IF cmd <> 0 AND lastCmd <> cmd and (((NOT strAI.opcCommandsDisabled) AND source > 0) OR source = 0) then
  	CASE BYTE_TO_INT(cmd) OF
  	(*cmd_SetUstavki*) 1 :
  				IF ((parametr AND _AnalogLimitFlags.LL) <> 0)		             	THEN 	strAI.LL := strAI.dLL; END_IF;
  				IF ((parametr AND _AnalogLimitFlags.HL) <> 0)		 	          THEN	strAI.HL := strAI.dHL; END_IF;
  				IF ((parametr AND _AnalogLimitFlags.LA) <> 0) AND strAI.ISVALIDREF_LA 	THEN	strAI.LA := strAI.dLA; END_IF;
  				IF ((parametr AND _AnalogLimitFlags.HA) <> 0) AND strAI.ISVALIDREF_HA 	THEN	strAI.HA := strAI.dHA; END_IF;
  				IF ((parametr AND _AnalogLimitFlags.LW) <> 0) AND strAI.ISVALIDREF_LW 	THEN	strAI.LW := strAI.dLW; END_IF;
  				IF ((parametr AND _AnalogLimitFlags.HW) <> 0) AND strAI.ISVALIDREF_HW 	THEN	strAI.HW := strAI.dHW; END_IF;
  	(*cmd_SetRemont*) 6 :
  				strAI.remont := TRUE;
  	(*cmd_ResetRemont*) 7 :
  				strAI.remont := FALSE;
  	(*cmd_kvitNotReliable*) 4 :
  				notReliable := FALSE;
  	END_CASE;
  	source_for_Status := source;
  	cmd_for_Status := cmd;
  	command_error_for_Status := 0;
  	resetCmdTimer(IN := FALSE);
  	resetCmdTimerPriznak := TRUE;
  END_IF;
  lastCmd := cmd;

  resetCmdTimer(IN := resetCmdTimerPriznak, PT := T#5S);
  IF resetCmdTimer.Q THEN
  	resetCmdTimerPriznak := FALSE;
  	source_for_Status := 0;
  	cmd_for_Status := 0;
  	command_error_for_Status := 0;
  END_IF;

  strAI.NS_Min := (strAI.value < strAI.minValue) AND strAI.minValue_ISVALIDREF;
  strAI.NS_Max := (strAI.value > strAI.maxValue) AND strAI.maxValue_ISVALIDREF;

  strAI.NS := (strAI.interval <= _statusAi.normal) AND NOT strAI.remont;

  Normal_trig(CLK := strAI.interval >= _statusAi.normal);

  IF NOT Normal_trig.Q THEN
  	_LastValueTimer(PT := T#1S);
  	IF (strAI.value<>_lastValue) OR _LastValueTimer.Q THEN
  		IF (_LastValueTimer.ET>T#0MS) THEN
  			strAI.ChangeSpeed:=(strAI.value-_lastValue)/(TIME_TO_LREAL(_LastValueTimer.ET));
  		END_IF;
  		_LastValueTimer(IN:=FALSE);

  		_LastValueTimer(IN:=TRUE);
  	END_IF;
  END_IF;
  _lastValue := strAI.value;

  IF ((strAI.maxChangeSpeed<>0.0) OR  (strAI.maxChangeSpeedDown<>0.0)) AND ( strAI.interval>=_statusAi.normal) THEN
  		IF (strAI.ChangeSpeed>0.0) THEN
  		    IF (strAI.ChangeSpeed > strAI.maxChangeSpeed) AND (strAI.maxChangeSpeed>0.0000001) THEN
  			 notReliable:=TRUE;
  		    END_IF;
  		ELSE
  		    IF (ABS(strAI.ChangeSpeed)>strAI.maxChangeSpeedDown) AND (strAI.maxChangeSpeedDown>0.0000001)  THEN
                                 notReliable:=TRUE;
  		    END_IF;
  		END_IF;

  END_IF;

  strAI.status := SHL(BYTE_TO_DWORD(source_for_Status), 29) 		              (* Источник команды *)
  			OR SHL(BYTE_TO_DWORD(cmd_for_Status), 26) 	    (* Команда *)
  			OR SHL(BYTE_TO_DWORD(command_error_for_Status), 23)   (* Ошибка команды *)
  			OR SHL(BOOL_TO_DWORD(strAI.OpcCommandsDisabled ), 21) (* Управление в ВУ заблокировано *)
  			OR SHL(BOOL_TO_DWORD(strAI.Disabled_HA), 9)		    (* ВА исключена из формирования интервала *)
  			OR SHL(BOOL_TO_DWORD(strAI.Disabled_LA), 8)		    (* НА исключена из формирования интервала *)
  			OR SHL(BOOL_TO_DWORD(strAI.Disabled_HW), 7)		    (* ВП исключена из формирования интервала *)
  			OR SHL(BOOL_TO_DWORD(strAI.Disabled_LW), 6)	              (* НП исключена из формирования интервала *)
  			OR SHL(BOOL_TO_DWORD(strAI.NS), 5)			    (* неиспарвность сигнала *)
  			OR SHL(BOOL_TO_DWORD(strAI.remont), 4)	              (* Выведен в ремонт *)
  			OR BYTE_TO_DWORD(strAI.interval);	              (* интервал *)
END_FUNCTION_BLOCK

FUNCTION_BLOCK Proc_Ai
  VAR
    fb_A1 : fb_AiSourceMlp;
    fb_A2 : fb_AiSourceMlp;
  END_VAR
  VAR_EXTERNAL
    Ai : AiConfig;
    arAIN_0 : TItemAIN;
    arAIN_1 : TItemAIN;
    AI_0_dblValue : LREAL;
    AI_1_dblValue : LREAL;
    arERR_0 : TItemDIN;
  END_VAR

  fb_A1(arAIN := arAIN_0, strAI := Ai.A1, err_mod := arERR_0);
  AI_0_dblValue := arAIN_0.dblValue;

  fb_A2(arAIN := arAIN_1, strAI := Ai.A2, err_mod := arERR_0);
  AI_1_dblValue := arAIN_1.dblValue;
END_FUNCTION_BLOCK

FUNCTION_BLOCK Opc_Ai_init
  VAR_EXTERNAL
    Ai : AiConfig;
    AI_A1_HW : LREAL;
    AI_A1_newHW : LREAL;
    AI_A1_HA : LREAL;
    AI_A1_newHA : LREAL;
    AI_A1_LA : LREAL;
    AI_A1_newLA : LREAL;
    AI_A1_LW : LREAL;
    AI_A1_newLW : LREAL;
    AI_A1_HL : LREAL;
    AI_A1_newHL : LREAL;
    AI_A1_LL : LREAL;
    AI_A1_newLL : LREAL;
    AI_A2_HW : LREAL;
    AI_A2_newHW : LREAL;
    AI_A2_HA : LREAL;
    AI_A2_newHA : LREAL;
    AI_A2_LA : LREAL;
    AI_A2_newLA : LREAL;
    AI_A2_LW : LREAL;
    AI_A2_newLW : LREAL;
    AI_A2_HL : LREAL;
    AI_A2_newHL : LREAL;
    AI_A2_LL : LREAL;
    AI_A2_newLL : LREAL;
  END_VAR

  AI_A1_HW := Ai.A1.HW;
  AI_A1_newHW := Ai.A1.dHW;
  AI_A1_HA := Ai.A1.HA;
  AI_A1_newHA := Ai.A1.dHA;
  AI_A1_LA := Ai.A1.LA;
  AI_A1_newLA := Ai.A1.dLA;
  AI_A1_LW := Ai.A1.LW;
  AI_A1_newLW := Ai.A1.dLW;
  AI_A1_LL := Ai.A1.LL;
  AI_A1_newLL := Ai.A1.dLL;
  AI_A1_HL := Ai.A1.HL;
  AI_A1_newHL := Ai.A1.dHL;

  AI_A2_HW := Ai.A2.HW;
  AI_A2_newHW := Ai.A2.dHW;
  AI_A2_HA := Ai.A2.HA;
  AI_A2_newHA := Ai.A2.dHA;
  AI_A2_LA := Ai.A2.LA;
  AI_A2_newLA := Ai.A2.dLA;
  AI_A2_LW := Ai.A2.LW;
  AI_A2_newLW := Ai.A2.dLW;
  AI_A2_LL := Ai.A2.LL;
  AI_A2_newLL := Ai.A2.dLL;
  AI_A2_HL := Ai.A2.HL;
  AI_A2_newHL := Ai.A2.dHL;
END_FUNCTION_BLOCK

FUNCTION_BLOCK Opc_Ai_get
  VAR_EXTERNAL
    Ai : AiConfig;
    AI_A1_newHW : LREAL;
    AI_A1_newHA : LREAL;
    AI_A1_newLA : LREAL;
    AI_A1_newLW : LREAL;
    AI_A1_newHL : LREAL;
    AI_A1_newLL : LREAL;
    AI_A1_command : UINT;
    AI_A2_newHW : LREAL;
    AI_A2_newHA : LREAL;
    AI_A2_newLA : LREAL;
    AI_A2_newLW : LREAL;
    AI_A2_newHL : LREAL;
    AI_A2_newLL : LREAL;
    AI_A2_command : UINT;
  END_VAR

  Ai.A1.dHW := AI_A1_newHW;
  Ai.A1.dHA := AI_A1_newHA;
  Ai.A1.dLA := AI_A1_newLA;
  Ai.A1.dLW := AI_A1_newLW;
  Ai.A1.dHL := AI_A1_newHL;
  Ai.A1.dLL := AI_A1_newLL;
  Ai.A1.inCommand_ARM := UINT_TO_WORD(AI_A1_command);

  Ai.A2.dHW := AI_A2_newHW;
  Ai.A2.dHA := AI_A2_newHA;
  Ai.A2.dLA := AI_A2_newLA;
  Ai.A2.dLW := AI_A2_newLW;
  Ai.A2.dHL := AI_A2_newHL;
  Ai.A2.dLL := AI_A2_newLL;
  Ai.A2.inCommand_ARM := UINT_TO_WORD(AI_A2_command);
END_FUNCTION_BLOCK

FUNCTION_BLOCK fb_DO_Init
  VAR_INPUT
    data_Ini : BOOL;
    imit : BOOL    := FALSE;
  END_VAR
  VAR_IN_OUT
    strDO : struct_DO;
  END_VAR
  VAR_OUTPUT
    Init : BOOL    := FALSE;
  END_VAR

  (*****            Функциональный блок переинициализации структуры-дескриптора канала дискретного ввода.            *****)
   Init := FALSE;

      IF data_Ini THEN                            (* Параметрам требуется переинициализация. *)
          strDO.imit       := imit;
          data_Ini:=FALSE;
          Init := TRUE;
      END_IF;
    IF Init THEN
  imit:=FALSE;
     END_IF;
END_FUNCTION_BLOCK

FUNCTION_BLOCK fb_Kran
  VAR_INPUT
    statOn : BOOL;
    statOff : BOOL;
    statOn_reliability : BOOL;
    statOff_reliability : BOOL;
  END_VAR
  VAR_IN_OUT
    strKr : struct_Kran;
  END_VAR
  VAR_INPUT
    inNs : TYPE_ReliableBit;
    inAccident : TYPE_ReliableBit;
    inAuto : TYPE_ReliableBit;
    inManual : TYPE_ReliableBit;
    inLocal : TYPE_ReliableBit;
    inDistance : TYPE_ReliableBit;
    inErrorPowerOff : TYPE_ReliableBit;
    inErrorBlock : TYPE_ReliableBit;
    inSo : TYPE_ReliableBit;
    inSz : TYPE_ReliableBit;
    inDp : TYPE_ReliableBit;
  END_VAR
  VAR
    onInit : BOOL    := FALSE;
    _statOn : BOOL;
    _statOff : BOOL;
    getSdvig : BOOL;
    lastOnStatus : BYTE;
    cmd : BYTE;
    source : BYTE;
    lastCmd : BYTE;
    source_for_Status : BYTE;
    cmd_for_Status : BYTE;
    command_error_for_Status : BYTE;
    _sunpackerCommand : fb_sunpackerCommand;
    _statusDualInput : TYPE_statusDualInput;
    _commandDualInput : TYPE_commandDualInput;
    _commandErrorTimer : BOOL;
    resetErrorTimer : BOOL;
    _changWithoutCommand : BOOL;
    BlockedOpenControl : BOOL;
    errorCMDTimer : TON;
    _errorReset : TON;
    sdvigReset : TON;
    continueHoldCommandTimer : TON;
    outputsSets : TOF;
    dP_Trig : R_TRIG;
    dP_Trig_reliability : R_TRIG;
    resetBlockedOpenControl_Trig : R_TRIG;
  END_VAR
  VAR_IN_OUT
    cmdOn : BOOL;
    cmdOff : BOOL;
  END_VAR

  IF NOT onInit THEN
  IF strKr.ISVALIDREF_cmdOn XOR strKr.ISVALIDREF_cmdOff THEN
  	IF 	strKr.ISVALIDREF_cmdOn THEN
  		lastCmd:= 2; (*baseCmdOff*)
  	ELSE
  		lastCmd:= 1; (*baseCmdOn*)
  	END_IF;
  END_IF;
  onInit:=TRUE;
  END_IF;

  (* ---- Если управление с ВУ заблокировано, то в ИМ передаем команду из алгоритма ---- *)
  IF strKr.inOpcCommandsDisabled THEN
  	strKr.inCommand := strKr.inCommand_Alg;
  ELSE (* иначе передаем команду с АРМа*)
  	strKr.inCommand := strKr.inCommand_ARM;
  END_IF;

  (* ---- Формирование состояния механизма ---- *)

  IF (strKr.ISVALIDREF_statOn) OR (strKr.ISVALIDREF_statOff) THEN
  	IF (strKr.ISVALIDREF_statOn) AND (strKr.ISVALIDREF_statOff) THEN
  	strKr.reliability:= statOn_reliability AND statOff_reliability;
  		_statOn  := statOn;
  		_statOff := statOff;
  	ELSIF (strKr.ISVALIDREF_statOn) THEN
                       strKr.reliability:= statOn_reliability;
  		_statOn  := statOn;
  		_statOff := NOT statOn;
  	ELSIF (strKr.ISVALIDREF_statOff) THEN
  		 strKr.reliability:= statOff_reliability;
  		_statOn  := NOT statOff;
  		_statOff :=statOff;
  	END_IF;

  	IF strKr.reliability THEN
  		IF _statOn AND NOT _statOff 		THEN 	strKr.onStatus := _statusDualInput.STATUS_ON;
  		ELSIF _statOff AND NOT _statOn 	THEN 	strKr.onStatus := _statusDualInput.Status_OFF;
  		ELSIF NOT _statOn AND NOT _statOff 	THEN 	strKr.onStatus := _statusDualInput.STATUS_TRANSITIONAL;
  		ELSE					strKr.onStatus := _statusDualInput.STATUS_ERROR;
                      END_IF;

  	ELSE
  		strKr.onStatus := _statusDualInput.STATUS_NOTDEFINED;

  	END_IF;
  ELSE
  	CASE BYTE_TO_INT(lastCmd) OF
  		(*baseCmdOn*)  1: strKr.onStatus  := _statusDualInput.STATUS_ON;
  		(*baseCmdOff*) 2: strKr.onStatus  := _statusDualInput.STATUS_OFF;

  	ELSE
  		 strKr.onStatus := _statusDualInput.STATUS_NOTDEFINED;

  	END_CASE;
  END_IF;

  strKr.Accident := inAccident.value AND inAccident.reliability;
  strKr.Ns := inNs.value AND inNs.reliability;
  strKr.Auto := inAuto.value AND inAuto.reliability;
  strKr.Manual := inManual.value AND inManual.reliability;
  strKr.Local := inLocal.value AND inLocal.reliability;
  strKr.Distance := inDistance.value AND inDistance.reliability;
  strKr.ErrorPowerOff := inErrorPowerOff.value AND inErrorPowerOff.reliability;
  strKr.ErrorBlock := inErrorBlock.value AND inErrorBlock.reliability;
  strKr.OpcCommandsDisabled := strKr.inOpcCommandsDisabled;

  (* ---- Формирование признака блокировки Открытия крана по высокому давлению ---- *)
  	IF strKr.ISVALIDREF_inDp THEN

  		strKr.Dp := NOT inDp.value AND inDp.reliability;

  		dP_Trig(CLK := strKr.Dp );
  		dP_Trig_reliability(CLK :=NOT inDp.reliability);

  		IF dP_Trig.Q OR dP_Trig_reliability.Q THEN
  			BlockedOpenControl := TRUE;
  		END_IF;
  		(* ---- автоматический сброс *)
  		resetBlockedOpenControl_Trig(CLK := (inDp.value) AND inDp.reliability);
  		IF resetBlockedOpenControl_Trig.Q THEN
  			BlockedOpenControl := FALSE;
  		END_IF;
  	ELSE
  		strKr.Dp  := FALSE;
  		BlockedOpenControl := FALSE;
  	END_IF;

  (* ---- Формирование признака сдвига ---- *)
  getSdvig := FALSE;
  IF (strKr.ISVALIDREF_cmdOn OR strKr.ISVALIDREF_cmdOff) AND NOT strKr.Local THEN
  	IF NOT (strKr.CmdOn OR strKr.CmdOff) THEN
  		IF (lastOnStatus <> strKr.onStatus AND
  		(strKr.onStatus <> _statusDualInput.STATUS_NOTDEFINED AND strKr.onStatus <> _statusDualInput.STATUS_ERROR) AND
  		(lastOnStatus <> _statusDualInput.STATUS_NOTDEFINED AND lastOnStatus <> _statusDualInput.STATUS_ERROR)) THEN
  			strKr.sdvig   := TRUE;
  		END_IF;
  	END_IF;
  END_IF;

  IF getSdvig THEN strKr.sdvig:= TRUE; END_IF;

  sdvigReset(IN:=strKr.sdvig, PT:=T#15S);

  IF sdvigReset.Q THEN strKr.sdvig:=FALSE; END_IF;

  lastOnStatus := strKr.onStatus;

  (* ---- Распаковка команды ---- *)
  _sunpackerCommand(command := strKr.inCommand);
  	cmd := _sunpackerCommand.cmd;
  	source := _sunpackerCommand.source;

  (* ---- Обработка команды ---- *)
  IF cmd <> 0 AND lastCmd <> cmd and (((NOT strKr.opcCommandsDisabled) AND source > 0) OR source = 0) then
  	CASE BYTE_TO_INT(cmd) OF
  	(*cmd_open*) 1 :
  			IF NOT BlockedOpenControl THEN
                                IF  strKr.ISVALIDREF_cmdOn THEN strKr.CmdOn := TRUE;
  				IF strKr.ISVALIDREF_cmdOff THEN strKr.CmdOff := FALSE; END_IF;
  			ELSIF  strKr.ISVALIDREF_cmdOff THEN strKr.CmdOff := FALSE;  END_IF;
  			errorCMDTimer(IN := false);

  			_commandErrorTimer := true;
  			strKr.lastCmdIsOn := true;
                                END_IF;
  	(*cmd_close*) 2 :
  			IF strKr.ISVALIDREF_cmdOff THEN strKr.CmdOff := TRUE;
  				IF strKr.ISVALIDREF_cmdOn THEN strKr.CmdOn := FALSE; END_IF;
  			ELSIF strKr.ISVALIDREF_cmdOn THEN strKr.CmdOn := FALSE; END_IF;
  			errorCMDTimer(IN := false);

  			_commandErrorTimer := true;
  			strKr.lastCmdIsOn := false;
  	(*cmd_reset*) 3 :   IF (strKr.ISVALIDREF_statOn) OR (strKr.ISVALIDREF_statOff) THEN
  			strKr.CmdOn := FALSE;
  			strKr.CmdOff := FALSE;
                                lastCmd := 0;
  			_commandErrorTimer := false;
  			strKr.lastCmdIsOn := false;
                                END_IF;

  	END_CASE;
  	source_for_Status := source;
  	cmd_for_Status := cmd;
  	command_error_for_Status := 0;
  END_IF;
  lastCmd := cmd;

  errorCMDTimer(In := _commandErrorTimer, PT :=T#90s);

  continueHoldCommandTimer(IN:=(strKr.onStatus = _statusDualInput.STATUS_ON) OR
  (strKr.onStatus = _statusDualInput.STATUS_OFF), PT:=strKr.continueHoldCommand);

  (* ---- алгоритм  для команды ВКЛючить ---- *)
  IF (strKr.onStatus = _statusDualInput.STATUS_ON) and strKr.lastCmdIsOn  then
  	IF strKr.ISVALIDREF_cmdOn AND strKr.ISVALIDREF_cmdOff then
            IF continueHoldCommandTimer.Q THEN
            strKr.cmdOn := false; END_IF;
            END_IF;
  	 errorCMDTimer(In := false);
  	 _commandErrorTimer := false;
  	 cmd_for_Status := 0;
  	 source_for_Status := 0;
  END_IF;

  (* ---- off ---- *)
  IF (strKr.onStatus = _statusDualInput.STATUS_OFF) and  (NOT strKr.lastCmdIsOn) then
  	IF strKr.ISVALIDREF_cmdOn AND strKr.ISVALIDREF_cmdOff then
            IF continueHoldCommandTimer.Q THEN
            strKr.cmdOff := false; END_IF;
            END_IF;
  	 errorCMDTimer(In := false);
  	 _commandErrorTimer := false;
  	 cmd_for_Status := 0;
  	 source_for_Status := 0;
  END_IF;

  (* ---- ошибка исполнения команды ---- *)
  if errorCMDTimer.Q and (cmd_for_Status <> 0) then
  	command_error_for_Status :=  cmd_for_Status;
  	_commandErrorTimer := false;
  	strKr.CmdOn := false;
  	strKr.CmdOff := false;
  	(*lastCmd := 0;*)
  END_IF;

  (* ---- сброс ошибки команды ---- *)
  strKr.CommandFault := command_error_for_Status <> 0;
  _errorReset(IN := command_error_for_Status <> 0, PT := T#5S);
  IF _errorReset.Q THEN
  	cmd_for_Status := 0;
  	source_for_Status := 0;
  	command_error_for_Status := 0;

  END_IF;

  outputsSets(in := (strKr.ISVALIDREF_cmdOn and strKr.cmdOn ) OR (strKr.ISVALIDREF_cmdOff and strKr.cmdOff), PT := T#2S);
  	IF NOT outputsSets.Q THEN
  		strKr.So := inSo._inversed AND inSo.reliability AND strKr.ISVALIDREF_inSo;
  		strKr.Sz := inSz._inversed AND inSz.reliability AND strKr.ISVALIDREF_inSz;
  	END_IF;

  cmdOn := strKr.cmdOn;
  cmdOff:= strKr.cmdOff;

  (* ---- формирование зашифрованного статуса для АРМа ---- *)
  strKr.status := shl(BYTE_TO_DWORD(source_for_Status), 29)
  		OR shl(BYTE_TO_DWORD(cmd_for_Status), 26)
  		OR shl(BYTE_TO_DWORD(command_error_for_Status), 23)
  		OR shl(bool_to_DWORD(strKr.sdvig), 22)
  		OR shl(bool_to_DWORD(strKr.OpcCommandsDisabled), 21)
                      OR shl(bool_to_DWORD(strKr.Dp), 14)
                      OR shl(BOOL_TO_DWORD(strKr.Sz), 13)
  		OR shl(BOOL_TO_DWORD(strKr.So), 12)
  		OR shl(BOOL_TO_DWORD(strKr.ErrorBlock), 11)
  		OR shl(BOOL_TO_DWORD(strKr.ErrorPowerOff), 10)
  		OR shl(BOOL_TO_DWORD(strKr.Manual), 8)
  		OR shl(BOOL_TO_DWORD(strKr.Auto), 7)
  		OR shl(BOOL_TO_DWORD(strKr.Distance), 6)
  		OR shl(BOOL_TO_DWORD(strKr.Local), 5)
  		OR shl(BOOL_TO_DWORD(strKr.Ns), 4)
                  	OR shl(BOOL_TO_DWORD(strKr.Accident ),3)
  		OR BYTE_TO_DWORD(strKr.onStatus);
END_FUNCTION_BLOCK

FUNCTION_BLOCK fb_OilPump
  VAR_INPUT
    statOn : BOOL;
    statOff : BOOL;
    statOn_reliability : BOOL;
    statOff_reliability : BOOL;
  END_VAR
  VAR_IN_OUT
    StrSw : struct_OilPump;
  END_VAR
  VAR_INPUT
    inNs : TYPE_ReliableBit;
    inAccident : TYPE_ReliableBit;
    inLocal : TYPE_ReliableBit;
    inDistance : TYPE_ReliableBit;
    inBreakCmdOn : TYPE_ReliableBit;
    inBreakCmdOff : TYPE_ReliableBit;
  END_VAR
  VAR
    onInit : BOOL    := FALSE;
    _statOn : BOOL;
    _statOff : BOOL;
    getSdvig : BOOL;
    lastOnStatus : BYTE;
    cmd : BYTE;
    source : BYTE;
    lastCmd : BYTE;
    source_for_Status : BYTE;
    cmd_for_Status : BYTE;
    command_error_for_Status : BYTE;
    _sunpackerCommand : fb_sunpackerCommand;
    _statusDualInput : TYPE_statusDualInput;
    _commandDualInput : TYPE_commandDualInput;
    _commandErrorTimer : BOOL;
    resetErrorTimer : BOOL;
    _changWithoutCommand : BOOL;
    errorCMDTimer : TON;
    sdvigReset : TON;
    _errorReset : TON;
    outputsSets : TOF;
  END_VAR
  VAR_IN_OUT
    cmdOn : BOOL;
    cmdOff : BOOL;
  END_VAR

  IF NOT onInit THEN
  IF StrSw.ISVALIDREF_cmdOn XOR StrSw.ISVALIDREF_cmdOff THEN
  	IF 	StrSw.ISVALIDREF_cmdOn THEN
  		lastCmd:= 2; (*baseCmdOff*)
  	ELSE
  		lastCmd:= 1; (*baseCmdOn*)
  	END_IF;
  END_IF;
  onInit:=TRUE;
  END_IF;

  (* ---- Если управление с ВУ заблокировано, то в ИМ передаем команду из алгоритма ---- *)
  IF StrSw.inOpcCommandsDisabled THEN
  	StrSw.inCommand := StrSw.inCommand_Alg;
  ELSE (* иначе передаем команду с АРМа*)
  	StrSw.inCommand := StrSw.inCommand_ARM;
  END_IF;

  (* ---- Формирование состояния механизма ---- *)

  IF (StrSw.ISVALIDREF_statOn) OR (StrSw.ISVALIDREF_statOff) THEN
  	IF (StrSw.ISVALIDREF_statOn) AND (StrSw.ISVALIDREF_statOff) THEN
  	StrSw.reliability:= statOn_reliability AND statOff_reliability;
  		_statOn  := statOn;
  		_statOff := statOff;
  	ELSIF (StrSw.ISVALIDREF_statOn) THEN
                       StrSw.reliability:= statOn_reliability;
  		_statOn  := statOn;
  		_statOff := NOT statOn;
  	ELSIF (StrSw.ISVALIDREF_statOff) THEN
  		 StrSw.reliability:= statOff_reliability;
  		_statOn  := NOT statOff;
  		_statOff :=statOff;
  	END_IF;

  	IF StrSw.reliability THEN
  		IF _statOn AND NOT _statOff 		THEN 	StrSw.onStatus := _statusDualInput.STATUS_ON;
  		ELSIF _statOff AND NOT _statOn 	THEN 	StrSw.onStatus := _statusDualInput.Status_OFF;
  		ELSIF NOT _statOn AND NOT _statOff 	THEN 	StrSw.onStatus := _statusDualInput.STATUS_TRANSITIONAL;
  		ELSE					StrSw.onStatus := _statusDualInput.STATUS_ERROR;
                      END_IF;

  	ELSE
  		StrSw.onStatus := _statusDualInput.STATUS_NOTDEFINED;

  	END_IF;
  ELSE
  	CASE BYTE_TO_INT(lastCmd) OF
  		(*baseCmdOn*) 1: StrSw.onStatus  := _statusDualInput.STATUS_ON;
  		(*baseCmdOff*) 2: StrSw.onStatus  := _statusDualInput.STATUS_OFF;

  	ELSE
  		 StrSw.onStatus := _statusDualInput.STATUS_NOTDEFINED;

  	END_CASE;
  END_IF;

  StrSw.Accident := inAccident.value AND inAccident.reliability;
  StrSw.Ns := inNs.value AND inNs.reliability;
  StrSw.Local := inLocal.value AND inLocal.reliability;
  StrSw.Distance := inDistance.value AND inDistance.reliability;
  StrSw.OpcCommandsDisabled := StrSw.inOpcCommandsDisabled;

  StrSw.Blocked:=StrSw.Accident OR StrSw.Local OR StrSw.breakCmdOn OR StrSw.breakCmdOff OR StrSw.inBlocked;

  StrSw.Rezervny:=NOT StrSw.Osnovnoy;

  (* ---- Формирование признака сдвига ---- *)

  getSdvig := FALSE;
  IF (StrSw.ISVALIDREF_cmdOn OR StrSw.ISVALIDREF_cmdOff) AND NOT StrSw.Local THEN
  	IF NOT (StrSw.CmdOn OR StrSw.CmdOff) THEN
                       IF (lastOnStatus <> StrSw.onStatus AND
  		(StrSw.onStatus <> _statusDualInput.STATUS_NOTDEFINED AND
                       StrSw.onStatus <> _statusDualInput.STATUS_ERROR)     AND
  		(lastOnStatus <> _statusDualInput.STATUS_NOTDEFINED   AND
                       lastOnStatus <> _statusDualInput.STATUS_ERROR))
                      THEN
  			getSdvig   := TRUE;
  		END_IF;
  	END_IF;
  END_IF;

  IF getSdvig THEN StrSw.sdvig:= TRUE; END_IF;

  sdvigReset(IN:=StrSw.sdvig, PT:=T#15S);

  IF sdvigReset.Q THEN StrSw.sdvig:=FALSE; END_IF;

  lastOnStatus := StrSw.onStatus;

  (* ---- Распаковка команды ---- *)
  _sunpackerCommand(command := StrSw.inCommand);
  	cmd := _sunpackerCommand.cmd;
  	source := _sunpackerCommand.source;

  (* ---- Обработка команды ---- *)
  IF cmd <> 0 AND lastCmd <> cmd and (((NOT StrSw.opcCommandsDisabled) AND source > 0) OR source = 0) then
  	CASE BYTE_TO_INT(cmd) OF
  	(*cmd_on*) 1 :
  			IF  StrSw.ISVALIDREF_cmdOn THEN StrSw.CmdOn := TRUE;
  				IF StrSw.ISVALIDREF_cmdOff THEN StrSw.CmdOff := FALSE; END_IF;
  			ELSIF  StrSw.ISVALIDREF_cmdOff THEN StrSw.CmdOff := FALSE;  END_IF;
  			errorCMDTimer(IN := false);
  			_commandErrorTimer := true;
  			StrSw.lastCmdIsOn := true;
  	(*cmd_off*) 2 :
  			IF StrSw.ISVALIDREF_cmdOff THEN StrSw.CmdOff := TRUE;
  				IF StrSw.ISVALIDREF_cmdOn THEN StrSw.CmdOn := FALSE; END_IF;
  			ELSIF StrSw.ISVALIDREF_cmdOn THEN StrSw.CmdOn := FALSE; END_IF;
  			errorCMDTimer(IN := false);

  			_commandErrorTimer := true;
  			StrSw.lastCmdIsOn := false;
  	(*cmd_reset*) 3 :    IF StrSw.ISVALIDREF_statOn OR StrSw.ISVALIDREF_statOff THEN
  			StrSw.CmdOn := FALSE;
  			StrSw.CmdOff := FALSE;
                                lastCmd := 0;
  			_commandErrorTimer := false;
  			StrSw.lastCmdIsOn := false;
                                 END_IF;
  	END_CASE;
  	source_for_Status := source;
  	cmd_for_Status := cmd;
  	command_error_for_Status := 0;
  END_IF;

  lastCmd := cmd;
  errorCMDTimer(In := _commandErrorTimer, PT :=T#10s);

  (* ---- алгоритм  для команды ВКЛючить ---- *)
  IF (StrSw.onStatus = _statusDualInput.STATUS_ON) and StrSw.lastCmdIsOn then
  	IF StrSw.ISVALIDREF_cmdOn AND StrSw.ISVALIDREF_cmdOff then  StrSw.cmdOn := false; END_IF;

  	 errorCMDTimer(In := false);
  	 _commandErrorTimer := false;
  	 cmd_for_Status := 0;
  	 source_for_Status := 0;
  END_IF;

  (* ---- off ---- *)
  IF (StrSw.onStatus = _statusDualInput.STATUS_OFF) and (NOT StrSw.lastCmdIsOn) then
  	IF StrSw.ISVALIDREF_cmdOn AND StrSw.ISVALIDREF_cmdOff then  StrSw.cmdOff := false; END_IF;

  	 errorCMDTimer(In := false);
  	 _commandErrorTimer := false;
  	 cmd_for_Status := 0;
  	 source_for_Status := 0;
  END_IF;

  (* ---- ошибка исполнения команды ---- *)
  if errorCMDTimer.Q and (cmd_for_Status <> 0) then
  	command_error_for_Status :=  cmd_for_Status;
  	_commandErrorTimer := false;
  	StrSw.CmdOn := false;
  	StrSw.CmdOff := false;
  	lastCmd := 0;
  end_if;

  (* ---- сброс ошибки команды ---- *)
  StrSw.CommandFault := command_error_for_Status <> 0;
  _errorReset(IN := command_error_for_Status <> 0, PT := T#5S);
  IF _errorReset.Q THEN
  	cmd_for_Status := 0;
  	source_for_Status := 0;
  	command_error_for_Status := 0;
  END_IF;

  outputsSets(in := (StrSw.ISVALIDREF_cmdOn and StrSw.cmdOn ) OR (StrSw.ISVALIDREF_cmdOff and StrSw.cmdOff), PT := T#2S);
  	IF NOT outputsSets.Q THEN
  		StrSw.BreakCmdOn := inBreakCmdOn._inversed AND inBreakCmdOn.reliability AND StrSw.ISVALIDREF_inBreakCmdOn;
  		StrSw.BreakCmdOff := inBreakCmdOff._inversed AND inBreakCmdOff.reliability AND StrSw.ISVALIDREF_inBreakCmdOff;
  	END_IF;

  cmdOn := StrSw.cmdOn;
  cmdOff:= StrSw.cmdOff;

  (* ---- формирование зашифрованного статуса для АРМа ---- *)
  StrSw.status := shl(BYTE_TO_DWORD(source_for_Status), 29)
  		OR shl(BYTE_TO_DWORD(cmd_for_Status), 26)
  		OR shl(BYTE_TO_DWORD(command_error_for_Status), 23)
  		OR shl(bool_to_DWORD(StrSw.sdvig), 22)
  		OR shl(bool_to_DWORD(StrSw.OpcCommandsDisabled), 21)
                      OR shl(bool_to_DWORD(StrSw.lastCmdIsOn), 14)
                      OR shl(BOOL_TO_DWORD(StrSw.BreakCmdOff), 13)
  		OR shl(BOOL_TO_DWORD(StrSw.BreakCmdOn), 12)
  		OR shl(BOOL_TO_DWORD(StrSw.Distance), 6)
  		OR shl(BOOL_TO_DWORD(StrSw.Local), 5)
  		OR shl(BOOL_TO_DWORD(StrSw.Ns), 4)
                  	OR shl(BOOL_TO_DWORD(StrSw.Accident ),3)
  		OR BYTE_TO_DWORD(StrSw.onStatus);
END_FUNCTION_BLOCK

FUNCTION_BLOCK fb_SectionSwitch
  VAR_INPUT
    statOn : BOOL;
    statOff : BOOL;
    statOn_reliability : BOOL;
    statOff_reliability : BOOL;
  END_VAR
  VAR_IN_OUT
    StrSw : struct_SectionSwitch;
  END_VAR
  VAR_INPUT
    basketRolledIn : TYPE_ReliableBit;
    basketRolledOut : TYPE_ReliableBit;
    basketTest : TYPE_ReliableBit;
    inNs : TYPE_ReliableBit;
    inoffKNA : TYPE_ReliableBit;
    inAccident : TYPE_ReliableBit;
    inLocal : TYPE_ReliableBit;
    inDistance : TYPE_ReliableBit;
    inBreakCmdOn : TYPE_ReliableBit;
    inBreakCmdOff : TYPE_ReliableBit;
  END_VAR
  VAR
    onInit : BOOL    := FALSE;
    _statOn : BOOL;
    _statOff : BOOL;
    getSdvig : BOOL;
    lastOnStatus : BYTE;
    cmd : BYTE;
    source : BYTE;
    lastCmd : BYTE;
    source_for_Status : BYTE;
    cmd_for_Status : BYTE;
    command_error_for_Status : BYTE;
    _basketRolledIn : TYPE_ReliableBit;
    _basketRolledOut : TYPE_ReliableBit;
    _basketTest : TYPE_ReliableBit;
    _sunpackerCommand : fb_sunpackerCommand;
    _statusDualInput : TYPE_statusDualInput;
    _statusBasket : TYPE_basketStats;
    _commandDualInput : TYPE_commandDualInput;
    _commandErrorTimer : BOOL;
    resetErrorTimer : BOOL;
    _changWithoutCommand : BOOL;
    errorCMDTimer : TON;
    _errorReset : TON;
    sdvigReset : TON;
    outputsSets : TOF;
  END_VAR
  VAR_IN_OUT
    cmdOn : BOOL;
    cmdOff : BOOL;
  END_VAR

  IF NOT onInit THEN
  IF StrSw.ISVALIDREF_cmdOn XOR StrSw.ISVALIDREF_cmdOff THEN
  	IF 	StrSw.ISVALIDREF_cmdOn THEN
  		lastCmd:= 2; (*baseCmdOff*)
  	ELSE
  		lastCmd:= 1; (*baseCmdOn*)
  	END_IF;
  END_IF;
  onInit:=TRUE;
  END_IF;

  (* ---- Формирование состояния тележки ---- *)

  IF (NOT StrSw.ISVALIDREF_basketRolledIn) AND (NOT StrSw.ISVALIDREF_basketRolledOut) THEN
            StrSw.basketStatus:=_statusBasket.BASKET_NOTDEFINED;
  ELSE
  		IF StrSw.ISVALIDREF_basketTest THEN
  		_basketTest:=basketTest;
  	ELSE
  		_basketTest.reliability:=TRUE;
  		_basketTest.value :=FALSE;
  	END_IF;

  	IF StrSw.ISVALIDREF_basketRolledIn THEN
  		_basketRolledIn:=basketRolledIn;
  	ELSE
  		_basketRolledIn:=basketRolledOut;
  		IF StrSw.ISVALIDREF_basketTest THEN
  		_basketRolledIn.value:=NOT (_basketRolledIn.value OR _basketTest.value);
  		ELSE
  		_basketRolledIn.value:= NOT _basketRolledIn.value;
  		END_IF;

  	END_IF;

  	IF StrSw.ISVALIDREF_basketRolledOut THEN
  		_basketRolledOut:=basketRolledOut;
  	ELSE
  		_basketRolledOut:=basketRolledIn;
  		IF StrSw.ISVALIDREF_basketTest THEN
  		_basketRolledOut.value:= NOT (_basketRolledOut.value OR _basketTest.value );
  		ELSE
  			_basketRolledOut.value := NOT _basketRolledout.value;
  		END_IF;

  	END_IF;

  IF _basketRolledIn.reliability AND _basketRolledOut.reliability AND _basketTest.reliability THEN
  		IF (BOOL_TO_INT(_basketRolledIn.value)+BOOL_TO_INT(_basketRolledOut.value)+BOOL_TO_INT(_basketTest.value))=1 THEN
  			IF _basketRolledIn.value THEN
  				StrSw.basketStatus:=_statusBasket.BASKET_ROLLEDIN;
  			ELSIF _basketRolledOut.value THEN
  				StrSw.basketStatus:=_statusBasket.BASKET_ROLLEDOUT;
  			ELSIF _basketTest.value THEN
  				StrSw.basketStatus:=_statusBasket.BASKET_TEST;
  			END_IF;
  		ELSE
  			StrSw.basketStatus:=_statusBasket.BASKET_ERROR;
  		END_IF;
  	ELSE
  		StrSw.basketStatus:=_statusBasket.BASKET_NOTDEFINED;
  	END_IF;
  END_IF;

  (* ---- Если управление с ВУ заблокировано, то в ИМ передаем команду из алгоритма ---- *)
  IF StrSw.inOpcCommandsDisabled THEN
  	StrSw.inCommand := StrSw.inCommand_Alg;
  ELSE (* иначе передаем команду с АРМа*)
  	StrSw.inCommand := StrSw.inCommand_ARM;
  END_IF;

  (* ---- Формирование состояния механизма ---- *)

  IF (StrSw.ISVALIDREF_statOn) OR (StrSw.ISVALIDREF_statOff) THEN
  	IF (StrSw.ISVALIDREF_statOn) AND (StrSw.ISVALIDREF_statOff) THEN
  	StrSw.reliability:= statOn_reliability AND statOff_reliability;
  		_statOn  := statOn;
  		_statOff := statOff;
  	ELSIF (StrSw.ISVALIDREF_statOn) THEN
                       StrSw.reliability:= statOn_reliability;
  		_statOn  := statOn;
  		_statOff := NOT statOn;
  	ELSIF (StrSw.ISVALIDREF_statOff) THEN
  		 StrSw.reliability:= statOff_reliability;
  		_statOn  := NOT statOff;
  		_statOff :=statOff;
  	END_IF;

  	IF StrSw.reliability THEN
  		IF _statOn AND NOT _statOff 		THEN 	StrSw.onStatus := _statusDualInput.STATUS_ON;
  		ELSIF _statOff AND NOT _statOn 	THEN 	StrSw.onStatus := _statusDualInput.Status_OFF;
  		ELSIF NOT _statOn AND NOT _statOff 	THEN 	StrSw.onStatus := _statusDualInput.STATUS_TRANSITIONAL;
  		ELSE					StrSw.onStatus := _statusDualInput.STATUS_ERROR;
                      END_IF;

  	ELSE
  		StrSw.onStatus := _statusDualInput.STATUS_NOTDEFINED;

  	END_IF;
  ELSE
  	CASE BYTE_TO_INT(lastCmd) OF
  		(*baseCmdOn*) 1: StrSw.onStatus  := _statusDualInput.STATUS_ON;
  		(*baseCmdOff*) 2: StrSw.onStatus  := _statusDualInput.STATUS_OFF;

  	ELSE
  		 StrSw.onStatus := _statusDualInput.STATUS_NOTDEFINED;
